// TwinCAT 3 PLC project M1_CompPP
// ProgramVersion: 3.1.4023.0
// libraries:
//   Tc2_Standard, * (Beckhoff Automation GmbH)
//   Tc2_System, * (Beckhoff Automation GmbH)
//   Tc2_Utilities, * (Beckhoff Automation GmbH)
//   Tc3_EventLogger, * (Beckhoff Automation GmbH)
//   Tc3_Module, * (Beckhoff Automation GmbH)
// project tree:
//   DUTs/ E_ChargerType.TcDUT, E_State.TcDUT, E_VoltFB.TcDUT, ST_Alarm_Base.TcDUT (not stored), ST_Charger_Base.TcDUT, ST_ChargeTime.TcDUT (not stored), ST_Module.TcDUT, ST_Segment_Base.TcDUT, ST_Setpoints_Base.TcDUT, ST_VoltMon_Base.TcDUT, ST_VoltTran_Base.TcDUT (not stored)
//   GVLs/ Alarms_DB.TcGVL (not stored), ChargeTime_DB.TcGVL, EngVal.TcGVL, GVL.TcGVL (not stored), HMI_DB.TcGVL, Input.TcGVL, LCP1_IO.TcGVL, LCP2_IO.TcGVL, LCP3_IO.TcGVL, LV.TcGVL, MCP_IO.TcGVL, Output.TcGVL, Permissives_DB.TcGVL, Setpoints.TcGVL, Trips_DB.TcGVL, VoltMonitor_DB.TcGVL
//   / PlcTask.TcTTO
//   POUs/ ADC_10V.TcPOU (not stored), ADC_5V.TcPOU (not stored), Alarms.TcPOU, Alarms_FB.TcPOU, Alias.TcPOU, AnalogConversion.TcPOU, AQ.TcPOU (not stored), ChargeTime.TcPOU, Heartbeat.TcPOU (not stored), HMI.TcPOU, LCA_CAL.TcPOU (not stored), MAIN.TcPOU, Norm_x.TcPOU (not stored), Permissives.TcPOU, Stagger_FB.TcPOU, Sequence.TcPOU, VoltageMonitor.TcPOU, VoltMonAC_FB.TcPOU, VoltTranBd.TcPOU (not stored)
// real-time tasks:
//   TASK PlcTask: cycle T#10ms, priority 20, ADS port 350
// I/O:
//   DEVICE Device 1 (EtherCAT) (disabled), AmsNetId 5.107.220.56.2.1
//     Term 1 (EK1200) [EK1200-5000 EtherCAT Power supply (2A E-Bus)]
//       Term 2 (EL1008) [EL1008 8Ch. Dig. Input 24V, 3ms]
//       Term 3 (EL6695) [EL6695 EtherCAT Bridge terminal (Primary)]
//       Term 4 (EK1561) [EK1561 1 port EtherCAT junction (POF)]
//       Term 5 (EL9011) [EL9011 End Terminal]

CONFIGURATION M1_CompPP
    RESOURCE PLC ON TwinCAT3
        TASK PlcTask(INTERVAL := T#10ms, PRIORITY := 20);
        PROGRAM MAIN WITH PlcTask : MAIN;
    END_RESOURCE
END_CONFIGURATION

// ---- DUTs/E_ChargerType.TcDUT
{attribute 'qualified_only'}
{attribute 'strict'}
TYPE E_ChargerType :
(
	TDK12kV := 0,
	TDK30kV := 1,
	TDK50kV := 2
);
END_TYPE

// ---- DUTs/E_State.TcDUT
{attribute 'qualified_only'}
{attribute 'strict'}
TYPE E_State :
(
	SAFE			:= 0, //IDLE
	CHARGING		:= 1, //Charge
	CHARGECOMPLETE	:= 2, //EOC
	//DISCONNECTING	:= 3, //Disconnect
	DUMPING			:= 3, 
	ABORT			:= 4,
	TRIPPED			:= 5, 
	ManualMode		:= 6
);
END_TYPE

// ---- DUTs/E_VoltFB.TcDUT
{attribute 'qualified_only'}
{attribute 'strict'}
TYPE E_VoltFB :
(
	seg1 := 1,
	seg2 := 2,
	seg3 := 3
);
END_TYPE

// ---- DUTs/ST_Charger_Base.TcDUT
TYPE ST_Charger_Base :
STRUCT
	//DI
	inhibited 		: BOOL;
	EndOfCharge 	: BOOL;
	HV_isON			: BOOL;
	OverTemp		: BOOL;
	InterlockOpen	: BOOL;
	LoadFaulted		: BOOL;
	SummaryFaulted	: BOOL;
	
	//DQ
	inhibit			: BOOL;
	HV_ON			: BOOL;
	
	//AI
	voltageFeedback_raw 	: INT;
	voltageFeedback_norm 	: REAL;
	voltageFeedback			: REAL;
	
	currentFeedback_raw 	: INT;
	currentFeedback_norm	: REAL;
	currentFeedback			: REAL;
	
	//AQ
	voltageSP_norm	: REAL;
	voltageSP		: REAL;
	voltageSP_raw	: INT; // setpoint output to field device.
	
	//Internal
	//ChargerType_50kV : BOOL;
	//ChargerType_12kV : BOOL;
	ChargerType		 : INT;
	LossInhibit		 : BOOL;
	LossHVON		 : BOOL;
	LossInhibitTON	 : TON;
	LossHVON_TON	 : TON;
	
	ChargeTime		: ST_ChargeTime;
END_STRUCT
END_TYPE

// ---- DUTs/ST_Module.TcDUT
TYPE ST_Module :
STRUCT
	DumpRly_close	: BOOL;
	
	VoltageFeedback : ARRAY[1..2] OF REAL;
	VoltageFeedback_norm : ARRAY[1..2] OF REAL;
	VoltageFeedback_raw : ARRAY[1..2] OF DINT;
	//VTB : ARRAY[1..2] OF ST_VoltTran_Base;  uncomment this for troubleshooting the bits in VoltageMonitor POU
END_STRUCT
END_TYPE

// ---- DUTs/ST_Segment_Base.TcDUT
TYPE ST_Segment_Base :
STRUCT
	Module : ARRAY [1..9] OF ST_Module;	
	
	CloseChargeRly	: BOOL;
	ChargeRly_close : BOOL;

	OpenModule1To3DumpRly : BOOL; //Open Module1To3DumpRly
	OpenModule4To6DumpRly : BOOL;
	OpenModule7To9DumpRly : BOOL;
	
	//ShortContactClose	: BOOL;

END_STRUCT
END_TYPE

// ---- DUTs/ST_Setpoints_Base.TcDUT
TYPE ST_Setpoints_Base :
STRUCT
	RequiredChargedV : REAL := 12;
	TotalCapacitance : REAL := 10; //uF - LOCAL ONLY, NOT FROM MAIN PLC - LoadCapacitance
	PSratedV		 : REAL := 50;
	wLCA			 : BOOL := TRUE;
	NumOfCharger	 : INT := 2;
	eChargerType		: E_ChargerType;
END_STRUCT
END_TYPE

// ---- DUTs/ST_VoltMon_Base.TcDUT
TYPE ST_VoltMon_Base :
STRUCT
	VTB : ARRAY[0..24] OF ST_VoltTran_Base;
	//Heartbeat : BOOL := 0;
	(*BateryLow  : ARRAY[0..24] OF BOOL := 0;
	//Channel	: USINT; //ST_AnalogCHSelection;
	VoltageReading_raw : ARRAY[0..24] OF INT; //custom board
	VoltageReading_norm : ARRAY[0..24] OF REAL;
	//VoltageReading	: ARRAY[0..15] OF REAL;
	//LoadMaxRatedV	: REAL := 13800; //-2k TO 35kV
	//LoadMinRatedV	: REAL := -1450; //Jake's lab result
//***************************************
	CapRaw : ARRAY[0..24] OF UINT;
	CapRawBIT : ARRAY[0..24] OF STRING;
	//CapRaw_DummySnap : ARRAY[0..24] OF UINT;
	CapRaw_Str : ARRAY[0..24] OF STRING;
	
	DataNull : ARRAY[0..24] OF BOOL := 0;
	//cunter for missing packets
	missedCTU : CTU;
	//ONS	: R_TRIG;
	missingCNT : WORD :=0;
	LossVoltTransBoard : ARRAY[0..24] OF BOOL := 0;
//**********************************	
	Time1		: TON;
	Time1_ET	: TIME;
	packetsPerMin : REAL;
	//missedCTU : CTU;
	ONS	: R_TRIG;
	//missingCNT : WORD;
	missingCNT_REAL : REAL;*)
END_STRUCT
END_TYPE

// ---- GVLs/ChargeTime_DB.TcGVL
{attribute 'qualified_only'}
VAR_GLOBAL RETAIN
	ChargerDelay_TON : ARRAY[1..7] OF TON;
	ChargerDelay_PT  : ARRAY[1..7] OF TIME;
	ChargerDelay_ET  : ARRAY[1..7] OF TIME;	
	
	//SustChargeTime_TON : ARRAY[1..3] OF TON;
	//SustChargeTime_PT  : ARRAY[1..3] OF TIME;
	//SustChargeTime_ET  : ARRAY[1..3] OF TIME;	
	
	//FormChargeTime_TON : ARRAY[1..2] OF TON;
	//FormChargeTime_PT  : ARRAY[1..2] OF TIME;
	//FormChargeTime_ET  : ARRAY[1..2] OF TIME;
	
	PreFormChargeTime_TON : TON;
	PreFormChargeTime_PT : TIME;
	PreFormChargeTime_ET : TIME;
	
	LongestChargeTime_TON : TON;
	LongestChargeTime_PT : TIME;
	LongestChargeTime_ET : TIME;

	ChargeTimeStartDelay	: ARRAY[1..7] OF INT;
	ChargingTimeElapse		: ARRAY[1..7] OF INT;	
	ChargingTimeElapse_TON	: ARRAY[1..7] OF TON;
	
	PreFormChargeTimeStartDelay : INT;
	PreFormChargingTimeElapse : INT;
	PreFormChargingTimeElapse_TON : TON;
END_VAR

// ---- GVLs/EngVal.TcGVL
{attribute 'qualified_only'}
VAR_GLOBAL
	Max_50kVChargerVoltage : REAL := 50000; //50kV
	Min_50kVChargerVoltage : REAL := 0;
	
	Max_50kVChargerCurrent : REAL := 0.18; //total peak charge current is 0.18A
	Min_50kVChargerCurrent : REAL := 0;
	
	Max_12kVChargerVoltage : REAL := 12000; //12kV
	Min_12kVChargerVoltage : REAL := 0;
	
	Max_12kVChargerCurrent : REAL := 0.75; //total peak charge current is 0.75A
	Min_12kVChargerCurrent : REAL := 0;
	
	Max_30kVChargerVoltage : REAL := 30000; //30kV
	Min_30kVChargerVoltage : REAL := 0;
	
	Max_30kVChargerCurrent : REAL := 0.6; //total peak charge current is 0.6A
	Min_30kVChargerCurrent : REAL := 0;	
	//Max_GLS1_ChargerV	   : REAL := 50000; //form trigger
	//Max_GLS2_ChargerV	   : REAL := 50000; // preform trigger
	//Max_GLS3_ChargerV	   : REAL := 30000; // preform cap charger
	
	Max_CapVoltage			: REAL := 32000;  //assuming 32kV cap....  
	Min_CapVoltage			: REAL := 0;
	
	UpperLimit12kVCaps		: REAL := 10500; 
	//LowerLimit12kVCaps	: REAL := -2000;
	UpperLimit50kVCaps		: REAL := 35000; 
	
	(*ULimit_PeakCapRequiredV	: REAL := 10000; //10kV veto
	LLimit_PeakCapRequiredV	: REAL := -2000; //-2kV
	ULimit_SustCapRequiredV	: REAL := 12000; //12kv veto
	LLimit_SustCapRequiredV	: REAL := -2000; //-2kv
	ULimit_FormCapRequiredV : REAL := 35000;
	LLimit_FormCapRequiredV : REAL := 0;
	*)
	//ULimit_PreFormCapRequiredV : REAL := 30000; //gls3
	//LLimit_PreFormCapRequiredV : REAL := 0;
		
END_VAR

// ---- GVLs/HMI_DB.TcGVL
{attribute 'qualified_only'}
VAR_GLOBAL PERSISTENT
	TDKLoad		: ARRAY [1..7] OF ST_Setpoints_Base; //or RETAIN
	
	ChargerHVOFF_rlyDelayPT		: TIME := T#25MS;
	ChargerHVOFF_rlyDelayPT_INT	: INT := 25;
	
	HVONdelayPT					: TIME := T#250MS;
	HVONdelayPT_INT				: INT := 250;
	
	RunOutTMR_PT				: TIME := T#10S;
	RunOutTMR_PT_INT			: DINT := 10;
	RunOutTMR_elapse			: DINT;
	
	ChargingRunOutTMR_elapse	: INT;

END_VAR

VAR_GLOBAL
	ChargePB					: BOOL := 0;
	DumpPB						: BOOL := 0;
	AbortPB						: BOOL := 0;
	FirePB						: BOOL := 0;
	ClearFaultPB				: BOOL := 0;
	AllDumpRelaysOpenBP			: BOOL := 0;
	AllDumpRelaysCloseBP		: BOOL := 0;
	AllCapsDischargedBP			: BOOL := 0;
	AllChargeRelayCloseBP		: BOOL := 0;
	AllVoltMonBoardStatusOKBP	: BOOL := 0;
	SystemSafeBP				: BOOL := 0;
	
	HMI_ManualModeSelected		: BOOL := 0;  // 1 = manual mode selected
	CloseChargeRlySW			: BOOL := 0;
	OpenDumpRlySW				: BOOL := 0;
	TurnChrgHVonSW				: BOOL := 0;
	TurnChrgInhibitOffSW		: BOOL := 0;
	TurnOnShotTrigSW			: BOOL := 0;
	TurnOnChargeAlarm			: BOOL := 0;
	
	LastTimeShotLog				: BOOL := 0;
END_VAR

// ---- GVLs/Input.TcGVL
{attribute 'qualified_only'}
VAR_GLOBAL
//***MCP************************************************************************
	//EL1008 - DI1
	R1_01_00 AT	%I*: BOOL; //Master stop PB not pressed - black pb on mcp
	R1_01_01 AT	%I*: BOOL; //case Estop circuit okay (Rly1 (120vac)
	R1_01_02 AT %I*: BOOL; //MCP PSU1 DC OK
	R1_01_03 AT %I*: BOOL; //
	R1_01_04 AT %I*: BOOL; //
	R1_01_05 AT %I*: BOOL; //spare
	R1_01_06 AT %I*: BOOL; //spare
	R1_01_07 AT %I*: BOOL; //spare

	//EL1008 - DI2
	R1_02_00 AT	%I*: BOOL; 
	R1_02_01 AT	%I*: BOOL;
	R1_02_02 AT %I*: BOOL; 
	R1_02_03 AT %I*: BOOL; 
	R1_02_04 AT %I*: BOOL; 
	R1_02_05 AT %I*: BOOL; 
	R1_02_06 AT %I*: BOOL; 
	R1_02_07 AT %I*: BOOL;  
	
	//EL1008 - DI3
	R1_03_00 AT	%I*: BOOL;  
	R1_03_01 AT	%I*: BOOL;
	R1_03_02 AT %I*: BOOL; 
	R1_03_03 AT %I*: BOOL; 
	R1_03_04 AT %I*: BOOL; 
	R1_03_05 AT %I*: BOOL; 
	R1_03_06 AT %I*: BOOL; 
	R1_03_07 AT %I*: BOOL;  
	
	//EL1008 - DI4
	R1_04_00 AT	%I*: BOOL;  
	R1_04_01 AT	%I*: BOOL;
	R1_04_02 AT %I*: BOOL; 
	R1_04_03 AT %I*: BOOL; 
	R1_04_04 AT %I*: BOOL; 
	R1_04_05 AT %I*: BOOL; 
	R1_04_06 AT %I*: BOOL; 
	R1_04_07 AT %I*: BOOL; 
	
	//EL1008 - DI5
	R1_05_00 AT	%I*: BOOL;  
	R1_05_01 AT	%I*: BOOL;
	R1_05_02 AT %I*: BOOL; 
	R1_05_03 AT %I*: BOOL; 
	R1_05_04 AT %I*: BOOL; 
	R1_05_05 AT %I*: BOOL; 
	R1_05_06 AT %I*: BOOL; 
	R1_05_07 AT %I*: BOOL;
	
	//EL3068 - AI1
	R1_08_00 		AT %I*: INT;
	R1_08_00_Status AT %I*: WORD;
	
	R1_08_01 		AT %I*: INT;
	R1_08_01_Status AT %I*: WORD;

	R1_08_02 		AT %I*: INT;
	R1_08_02_Status AT %I*: WORD;

	R1_08_03 		AT %I*: INT;
	R1_08_03_Status AT %I*: WORD;

	R1_08_04 		AT %I*: INT;
	R1_08_04_Status AT %I*: WORD;

	R1_08_05 		AT %I*: INT;
	R1_08_05_Status AT %I*: WORD;

	R1_08_06 		AT %I*: INT;
	R1_08_06_Status AT %I*: WORD;

	R1_08_07 		AT %I*: INT;
	R1_08_07_Status AT %I*: WORD;

//RACK 2
	//EL3068 - AI1
	R2_01_00 		AT %I*: INT;
	R2_01_00_Status AT %I*: WORD;

	R2_01_01 		AT %I*: INT;
	R2_01_01_Status AT %I*: WORD;

	R2_01_02 		AT %I*: INT;
	R2_01_02_Status AT %I*: WORD;

	R2_01_03 		AT %I*: INT;
	R2_01_03_Status AT %I*: WORD;

	R2_01_04 		AT %I*: INT;
	R2_01_04_Status AT %I*: WORD;

	R2_01_05 		AT %I*: INT;
	R2_01_05_Status AT %I*: WORD;

	R2_01_06 		AT %I*: INT;
	R2_01_06_Status AT %I*: WORD;

	R2_01_07 		AT %I*: INT;
	R2_01_07_Status AT %I*: WORD;

	//EL3068 - AI2
	R2_02_00 		AT %I*: INT;
	R2_02_00_Status AT %I*: WORD;

	R2_02_01 		AT %I*: INT;
	R2_02_01_Status AT %I*: WORD;

	R2_02_02 		AT %I*: INT;
	R2_02_02_Status AT %I*: WORD;

	R2_02_03 		AT %I*: INT;
	R2_02_03_Status AT %I*: WORD;

	R2_02_04 		AT %I*: INT;
	R2_02_04_Status AT %I*: WORD;

	R2_02_05 		AT %I*: INT;
	R2_02_05_Status AT %I*: WORD;

	R2_02_06 		AT %I*: INT;
	R2_02_06_Status AT %I*: WORD;

	R2_02_07 		AT %I*: INT;
	R2_02_07_Status AT %I*: WORD;

	//EL1008 - DI1
	R2_03_00 AT	%I*: BOOL;  
	R2_03_01 AT	%I*: BOOL;
	R2_03_02 AT %I*: BOOL; 
	R2_03_03 AT %I*: BOOL; 
	R2_03_04 AT %I*: BOOL; 
	R2_03_05 AT %I*: BOOL; 
	R2_03_06 AT %I*: BOOL; 
	R2_03_07 AT %I*: BOOL;  

	//EL1008 - DI2
	R2_04_00 AT	%I*: BOOL;  
	R2_04_01 AT	%I*: BOOL;
	R2_04_02 AT %I*: BOOL; 
	R2_04_03 AT %I*: BOOL; 
	R2_04_04 AT %I*: BOOL; 
	R2_04_05 AT %I*: BOOL; 
	R2_04_06 AT %I*: BOOL; 
	R2_04_07 AT %I*: BOOL;  

	//EL1008 - DI3
	R2_05_00 AT	%I*: BOOL;  
	R2_05_01 AT	%I*: BOOL;
	R2_05_02 AT %I*: BOOL; 
	R2_05_03 AT %I*: BOOL; 
	R2_05_04 AT %I*: BOOL; 
	R2_05_05 AT %I*: BOOL; 
	R2_05_06 AT %I*: BOOL; 
	R2_05_07 AT %I*: BOOL;  

//Rack 3	
	//EL3068 - AI1
	R3_01_00 		AT %I*: INT;
	R3_01_00_Status AT %I*: WORD;

	R3_01_01 		AT %I*: INT;
	R3_01_01_Status AT %I*: WORD;

	R3_01_02 		AT %I*: INT;
	R3_01_02_Status AT %I*: WORD;

	R3_01_03 		AT %I*: INT;
	R3_01_03_Status AT %I*: WORD;

	R3_01_04 		AT %I*: INT;
	R3_01_04_Status AT %I*: WORD;

	R3_01_05 		AT %I*: INT;
	R3_01_05_Status AT %I*: WORD;

	R3_01_06 		AT %I*: INT;
	R3_01_06_Status AT %I*: WORD;

	R3_01_07 		AT %I*: INT;
	R3_01_07_Status AT %I*: WORD;

	//EL3068 - AI2
	R3_02_00 		AT %I*: INT;
	R3_02_00_Status AT %I*: WORD;

	R3_02_01 		AT %I*: INT;
	R3_02_01_Status AT %I*: WORD;

	R3_02_02 		AT %I*: INT;
	R3_02_02_Status AT %I*: WORD;

	R3_02_03 		AT %I*: INT;
	R3_02_03_Status AT %I*: WORD;

	R3_02_04 		AT %I*: INT;
	R3_02_04_Status AT %I*: WORD;

	R3_02_05 		AT %I*: INT;
	R3_02_05_Status AT %I*: WORD;

	R3_02_06 		AT %I*: INT;
	R3_02_06_Status AT %I*: WORD;

	R3_02_07 		AT %I*: INT;
	R3_02_07_Status AT %I*: WORD;

	//EL1008 - DI1
	R3_03_00 AT	%I*: BOOL;  
	R3_03_01 AT	%I*: BOOL;
	R3_03_02 AT %I*: BOOL; 
	R3_03_03 AT %I*: BOOL; 
	R3_03_04 AT %I*: BOOL; 
	R3_03_05 AT %I*: BOOL; 
	R3_03_06 AT %I*: BOOL; 
	R3_03_07 AT %I*: BOOL;  

	//EL1008 - DI2
	R3_04_00 AT	%I*: BOOL;  
	R3_04_01 AT	%I*: BOOL;
	R3_04_02 AT %I*: BOOL; 
	R3_04_03 AT %I*: BOOL; 
	R3_04_04 AT %I*: BOOL; 
	R3_04_05 AT %I*: BOOL; 
	R3_04_06 AT %I*: BOOL; 
	R3_04_07 AT %I*: BOOL;  

	//EL1008 - DI3
	R3_05_00 AT	%I*: BOOL;  
	R3_05_01 AT	%I*: BOOL;
	R3_05_02 AT %I*: BOOL; 
	R3_05_03 AT %I*: BOOL; 
	R3_05_04 AT %I*: BOOL; 
	R3_05_05 AT %I*: BOOL; 
	R3_05_06 AT %I*: BOOL; 
	R3_05_07 AT %I*: BOOL; 
	
	//Ethercat Device Voltage - subject to change because the VM board is still under development
	B170357_CapRaw AT %I* : ARRAY[0..24] OF UINT;
	B170357_BatLevel AT %I* : BOOL;
	B170357_Heartbeat AT %I* : BOOL;
	
	B170357_2_CapRaw AT %I* : ARRAY[0..24] OF UINT;
	B170357_2_BatLevel AT %I* : BOOL;
	B170357_2_Heartbeat AT %I* : BOOL;
	
	//Ract 4 - Shaft ramp
	//EL1008 - DI 1
	R4_01_00 AT %I*: BOOL; 
	R4_01_01 AT	%I*: BOOL;
	R4_01_02 AT %I*: BOOL; 
	R4_01_03 AT %I*: BOOL; 
	R4_01_04 AT %I*: BOOL; 
	R4_01_05 AT %I*: BOOL; 
	R4_01_06 AT %I*: BOOL; 
	R4_01_07 AT %I*: BOOL; 
	
	B170357_3_CapRaw AT %I* : ARRAY[0..24] OF UINT;  // might be 8 fruit stands so 0..7
	B170357_3_BatLevel AT %I* : BOOL;
	B170357_3_Heartbeat AT %I* : BOOL;
	
END_VAR

// ---- GVLs/LCP1_IO.TcGVL
{attribute 'qualified_only'}
VAR_GLOBAL
	Segment	: ARRAY [1..3] OF ST_Segment_Base;
	
	Segment1to3_ShortContactClose	: BOOL;
	Segment1to3_UnShortContactClose	: BOOL;
	LossInterlockPressure			: BOOL;
	PSU1OK							: BOOL;
	
	VMB : ST_VoltMon_Base;
	//VTB : ARRAY[0..17] OF ST_VoltTran_Base; 
	Fire			: BOOL;
	SegmentCharged	: BOOL;
	TriggerScope	: BOOL;
END_VAR

// ---- GVLs/LCP2_IO.TcGVL
{attribute 'qualified_only'}
VAR_GLOBAL
	Segment	: ARRAY [4..6] OF ST_Segment_Base;
	
	Segment4to6_ShortContactClose	: BOOL;
	Segment4to6_UnShortContactClose	: BOOL;
	LossInterlockPressure			: BOOL;
	PSU1OK							: BOOL;
	
	VMB : ST_VoltMon_Base;
	Fire			: BOOL;
	SegmentCharged	: BOOL;
	TriggerScope	: BOOL;
END_VAR

// ---- GVLs/LCP3_IO.TcGVL
{attribute 'qualified_only'}
VAR_GLOBAL
	//Shaft Ramp Supply
	PSU1_OK				: BOOL := FALSE;
	VMB 				: ST_VoltMon_Base;
	SegmentCharged		: BOOL := FALSE;
	CloseSRChargeRly	: BOOL := FALSE;
	SRChargeRly_close 	: BOOL := FALSE;
	OpenSRDumpRly		: ARRAY[1..8] OF BOOL;
	SRDumpRelay_close 	: BOOL := FALSE;
END_VAR

// ---- GVLs/LV.TcGVL
{attribute 'qualified_only'}
VAR_GLOBAL
	TxWord1	: WORD;
	TxWord2 : WORD;
	TxWord3 : WORD;
	
	RxWord1 : WORD;
	RxWord2 : WORD;
	RxWord3 : WORD;

	
	TxInt : ARRAY [1..5] OF INT;
	TxDint : ARRAY [1..3] OF DINT;
	TxREAL : ARRAY [1..6] OF REAL;

	RxInt : ARRAY [1..2] OF INT;
	RxDint : ARRAY [1..3] OF DINT;
	RxREAL : ARRAY [1..44] OF REAL;
	
	Charger : ARRAY[1..6] OF ST_Charger_Base;
	
	TDKLoad	: ARRAY [1..6] OF ST_Setpoints_Base; 
	
	(*ChargerHVOFF_rlyDelayPT		: TIME := T#25MS;
	ChargerHVOFF_rlyDelayPT_INT	: INT := 25;
	
	HVONdelayPT					: TIME := T#250MS;
	HVONdelayPT_INT				: INT := 250;
	
	RunOutTMR_PT				: TIME := T#10S;
	RunOutTMR_PT_INT			: DINT := 10;
	RunOutTMR_elapse			: DINT;
	
	ChargingRunOutTMR_elapse	: INT;
	
	ChargePB					: BOOL := 0;
	DumpPB						: BOOL := 0;
	AbortPB						: BOOL := 0;
	FirePB						: BOOL := 0;
	ClearFaultPB				: BOOL := 0;
	AllDumpRelaysOpenBP			: BOOL := 0;
	AllChargeRelayCloseBP		: BOOL := 0;
	SystemSafeBP				: BOOL := 0;
	
	HMI_ManualModeSelected		: BOOL := 0;  // 1 = manual mode selected
	CloseChargeRlySW			: BOOL := 0;
	OpenDumpRlySW				: BOOL := 0;*)
END_VAR

// ---- GVLs/MCP_IO.TcGVL
{attribute 'qualified_only'}
VAR_GLOBAL
	MasterStopPB_NotPressed		: BOOL;
	CageEstopCircuitOK			: BOOL;
	//RemoteModeSelected			: BOOL;
	PSU1_DCOK					: BOOL;
	//MachineGNDrlyOpen			: BOOL;
	//CloseAllChargeRlyCommand	: BOOL; only for slim
	//OpenAllDumpRelayCommand		: BOOL; only for slim
	//Charger 					: ARRAY [1..8] OF ST_Charger_Base;
	//GLS3_Load					: ST_ChargeTime;
	//GLS1_hvON					: BOOL;
	//GLS2_hvON					: BOOL;
	//GLS3_hvON					: BOOL;
	//LiftMachineGND				: BOOL;
	//AllChargeRelaysClose		: BOOL; only for slim
	//AllDumpRelaysOpen			: BOOL; only for slim
	//GLS1_voltageSP				: DINT;
	//GLS1_voltageSP_norm			: REAL;
	//GLS1_voltageSP_raw			: INT;
	
	//GLS2_voltageSP				: DINT;
	//GLS2_voltageSP_norm			: REAL;
	//GLS2_voltageSP_raw			: INT;
	
	//GLS3_voltageSP				: DINT;
	//GLS3_voltageSP_norm			: REAL;
	//GLS3_voltageSP_raw			: INT;

END_VAR

VAR_GLOBAL PERSISTENT
	Charger 					: ARRAY [1..7] OF ST_Charger_Base;
END_VAR

// ---- GVLs/Output.TcGVL
{attribute 'qualified_only'}
VAR_GLOBAL
//***MCP 
	//EL2008 - DQ1
	R1_06_00 AT %Q*: BOOL;
	R1_06_01 AT %Q*: BOOL;
	R1_06_02 AT %Q*: BOOL;
	R1_06_03 AT %Q*: BOOL;
	R1_06_04 AT %Q*: BOOL;
	R1_06_05 AT %Q*: BOOL;
	R1_06_06 AT %Q*: BOOL;
	R1_06_07 AT %Q*: BOOL;

	//EL2008 - DQ2
	R1_07_00 AT %Q*: BOOL;
	R1_07_01 AT %Q*: BOOL;
	R1_07_02 AT %Q*: BOOL;
	R1_07_03 AT %Q*: BOOL;
	R1_07_04 AT %Q*: BOOL;
	R1_07_05 AT %Q*: BOOL;
	R1_07_06 AT %Q*: BOOL;
	R1_07_07 AT %Q*: BOOL;
	
	//EL4008 - AQ1
	R1_09_00 AT %Q*: INT;	//Charger 1 - Voltage Setpoint
	R1_09_01 AT %Q*: INT;	//Charger 2 - Voltage Setpoint
	R1_09_02 AT %Q*: INT;	//Charger 3 - Voltage Setpoint
	R1_09_03 AT %Q*: INT;	//Charger 4 - Voltage Setpoint
	R1_09_04 AT %Q*: INT;	//Charger 5 - Voltage Setpoint	
	R1_09_05 AT %Q*: INT;	//Charger 6 - Voltage Setpoint	
	R1_09_06 AT %Q*: INT;	//spare
	R1_09_07 AT %Q*: INT;	//spare
	
//**LCP1
	//EL2008 - DQ1
	R2_06_00 AT %Q*: BOOL;
	R2_06_01 AT %Q*: BOOL;
	R2_06_02 AT %Q*: BOOL;
	R2_06_03 AT %Q*: BOOL;
	R2_06_04 AT %Q*: BOOL;
	R2_06_05 AT %Q*: BOOL;
	R2_06_06 AT %Q*: BOOL;
	R2_06_07 AT %Q*: BOOL;
	
	//EL2008 - DQ2
	R2_07_00 AT %Q*: BOOL;
	R2_07_01 AT %Q*: BOOL;
	R2_07_02 AT %Q*: BOOL;
	R2_07_03 AT %Q*: BOOL;
	R2_07_04 AT %Q*: BOOL;
	R2_07_05 AT %Q*: BOOL;
	R2_07_06 AT %Q*: BOOL;
	R2_07_07 AT %Q*: BOOL;

//**LCP2
	//EL2008 - DQ1
	R3_06_00 AT %Q*: BOOL;
	R3_06_01 AT %Q*: BOOL;
	R3_06_02 AT %Q*: BOOL;
	R3_06_03 AT %Q*: BOOL;
	R3_06_04 AT %Q*: BOOL;
	R3_06_05 AT %Q*: BOOL;
	R3_06_06 AT %Q*: BOOL;
	R3_06_07 AT %Q*: BOOL;
	
	//EL2008 - DQ2
	R3_07_00 AT %Q*: BOOL;
	R3_07_01 AT %Q*: BOOL;
	R3_07_02 AT %Q*: BOOL;
	R3_07_03 AT %Q*: BOOL;
	R3_07_04 AT %Q*: BOOL;
	R3_07_05 AT %Q*: BOOL;
	R3_07_06 AT %Q*: BOOL;
	R3_07_07 AT %Q*: BOOL;
	
//**LCP3
	//EL2008 - DQ 1
	R4_02_00 AT %Q*: BOOL; 
	R4_02_01 AT	%Q*: BOOL; 
	R4_02_02 AT %Q*: BOOL; 
	R4_02_03 AT %Q*: BOOL; 
	R4_02_04 AT %Q*: BOOL; 
	R4_02_05 AT %Q*: BOOL; 
	R4_02_06 AT %Q*: BOOL; 
	R4_02_07 AT %Q*: BOOL; 
	//EL2008 - DQ2
	R4_03_00 AT %Q*: BOOL; 
	R4_03_01 AT	%Q*: BOOL; 
	R4_03_02 AT %Q*: BOOL; 
	R4_03_03 AT %Q*: BOOL; 
	R4_03_04 AT %Q*: BOOL; 
	R4_03_05 AT %Q*: BOOL; 
	R4_03_06 AT %Q*: BOOL; 
	R4_03_07 AT %Q*: BOOL; 	
END_VAR

// ---- GVLs/Permissives_DB.TcGVL
{attribute 'qualified_only'}
VAR_GLOBAL
	//SafetyOK				: BOOL;
	AllChargeRelayClosed 	: BOOL := 0;
	AllDumpRelayOpen		: BOOL := 0;
	//AllDumpRelayClose		: BOOL := 0;
	ReadyToCharge			: BOOL := 0;
	AllChargerEOC			: BOOL := 0;
	
	ChargerVBelowThres		: BOOL := 0;
	ChargerVThres			: REAL := 40;
	AllChargerHVisOFF		: BOOL := 0;
	AllChargerInhibitON		: BOOL := 0;

	AllCapsDischarged		: BOOL := 0;
	CapVoltageThres			: REAL := 40;
	
	AnyLCP1MonBoardLoss		: BOOL := 0;
	AnyLCP1MonBoardBatLo	: BOOL := 0;
	AnyLCP2MonBoardLoss		: BOOL := 0;
	AnyLCP2MonBoardBatLo	: BOOL := 0;
	
	AnyVoltMonBoardLoss		: BOOL := 0;
	AnyVoltMonBoardBatLo	: BOOL := 0;
	AllVoltMonBoardStatusOK : BOOL := 0;
	SystemIsSafe			: BOOL := 0;
END_VAR

// ---- GVLs/Setpoints.TcGVL
{attribute 'qualified_only'}
VAR_GLOBAL
	TDKLoad : ARRAY [1..7] OF ST_Setpoints_Base;
	
END_VAR

// ---- GVLs/Trips_DB.TcGVL
{attribute 'qualified_only'}
VAR_GLOBAL
		
	AnyEstopPressed 			: BOOL; //might not need
	MasterSTOPPressed			: BOOL;
	AllDCpsuOK					: BOOL;
	CageDoorNotClose			: BOOL; // might not need
	//AnyChargerOverTemp			: BOOL;
	//AnyChargerLoadFault			: BOOL;
	//AnyChargerInterlockOpen		: BOOL;
	//AnyChargerFaulted			: BOOL; // same as summary fault
	
	//SystemTripped 				: BOOL;
	//InstrumentationFaulted		: BOOL;
	//AnyChargeRlyFail			: BOOL;
	//AnyDumpRlyFail				: BOOL;
	//AnyACInterlockFail			: BOOL;
	//AnyLossInhibitSignal		: BOOL;
	//AnyLossHVONsignal			: BOOL;
	
	ChargingTimerRunout         : BOOL;
	ChargedTimerRunout			: BOOL;
	DumpTimerRunout				: BOOL;
	//SystemTimeOut				: BOOL;
	NoFaultDetected				: BOOL;
	TimerRunOutON				: BOOL;
	ChargerSummaryFault			: BOOL;
	ShortingSystemUnknown		: BOOL;
END_VAR

// ---- GVLs/VoltMonitor_DB.TcGVL
{attribute 'qualified_only'}
VAR_GLOBAL
	//VoltMonDB : ARRAY [1..2] OF ST_VoltMon_Base; 
END_VAR

// ---- POUs/MAIN.TcPOU
PROGRAM MAIN
VAR
END_VAR

Alias();
Permissives();
ChargeTime();
AnalogConversion();
VoltageMonitor();
Sequence();
HMI();
Alarms();
Heartbeat();

END_PROGRAM

// ---- POUs/Alias.TcPOU
PROGRAM Alias
VAR
	i : INT := 1;
	n : INT := 7;
	a : INT := 0; //0-15
	k : INT := 0;
	m : INT := 0;
	p : INT := 0;
END_VAR

//R1 : MCP**  
	//INPUT
	//DI
	MCP_IO.MasterStopPB_NotPressed				:= Input.R1_01_00;  //NC - Master stop PB not pressed - black pb on mcp
	MCP_IO.CageEstopCircuitOK					:= Input.R1_01_01;  //case Estop circuit okay (Rly1 (120vac)  
	MCP_IO.PSU1_DCOK							:= Input.R1_01_02; // psu1 dc ok
	//Spare										:= Input.R1_01_03; //
	//Spare										:= Input.R1_01_04; // 
	//Spare										:= Input.R1_01_05; //  
	//Spare										:= Input.R1_01_06; //  
	//Spare										:= Input.R1_01_07; //
	
	//DI
	MCP_IO.Charger[1].inhibited					:= NOT Input.R1_02_00; //TDK802 1
	MCP_IO.Charger[1].EndOfCharge				:= NOT Input.R1_02_01; //TDK802 1
	MCP_IO.Charger[1].HV_isON					:= NOT Input.R1_02_02; //TDK802 1
	MCP_IO.Charger[1].SummaryFaulted			:= NOT Input.R1_02_03; //TDK802 1
	MCP_IO.Charger[2].inhibited					:= NOT Input.R1_02_04; //TDK802 2
	MCP_IO.Charger[2].EndOfCharge				:= NOT Input.R1_02_05; //TDK802 2
	MCP_IO.Charger[2].HV_isON					:= NOT Input.R1_02_06; //TDK802 2
	MCP_IO.Charger[2].SummaryFaulted			:= NOT Input.R1_02_07; //TDK802 2
	
	MCP_IO.Charger[3].inhibited					:= NOT Input.R1_03_00; //TDK802 3
	MCP_IO.Charger[3].EndOfCharge				:= NOT Input.R1_03_01; //TDK802 3
	MCP_IO.Charger[3].HV_isON					:= NOT Input.R1_03_02; //TDK802 3
	MCP_IO.Charger[3].SummaryFaulted			:= NOT Input.R1_03_03; //TDK802 3
	MCP_IO.Charger[4].inhibited					:= NOT Input.R1_03_04; //TDK802 4
	MCP_IO.Charger[4].EndOfCharge				:= NOT Input.R1_03_05; //TDK802 4
	MCP_IO.Charger[4].HV_isON					:= NOT Input.R1_03_06; //TDK802 4
	MCP_IO.Charger[4].SummaryFaulted			:= NOT Input.R1_03_07; //TDK802 4
	
	MCP_IO.Charger[5].inhibited					:= NOT Input.R1_04_00; //TDK802 5
	MCP_IO.Charger[5].EndOfCharge				:= NOT Input.R1_04_01; //TDK802 5
	MCP_IO.Charger[5].HV_isON					:= NOT Input.R1_04_02; //TDK802 5
	MCP_IO.Charger[5].SummaryFaulted			:= NOT Input.R1_04_03; //TDK802 5
	MCP_IO.Charger[6].inhibited					:= NOT Input.R1_04_04; //TDK802 6
	MCP_IO.Charger[6].EndOfCharge				:= NOT Input.R1_04_05; //TDK802 6
	MCP_IO.Charger[6].HV_isON					:= NOT Input.R1_04_06; //TDK802 6
	MCP_IO.Charger[6].SummaryFaulted			:= NOT Input.R1_04_07; //TDK802 6
	(*shaft ramp add below*)
	
	//DQ
	Output.R1_06_00	:= MCP_IO.Charger[1].inhibit;
	Output.R1_06_01	:= MCP_IO.Charger[1].HV_ON;
	Output.R1_06_02	:= MCP_IO.Charger[2].inhibit;
	Output.R1_06_03	:= MCP_IO.Charger[2].HV_ON;
	Output.R1_06_04	:= MCP_IO.Charger[3].inhibit;
	Output.R1_06_05	:= MCP_IO.Charger[3].HV_ON;
	Output.R1_06_06	:= MCP_IO.Charger[4].inhibit;
	Output.R1_06_07	:= MCP_IO.Charger[4].HV_ON;
	
	//DQ
	Output.R1_07_00	:= MCP_IO.Charger[5].inhibit;
	Output.R1_07_01	:= MCP_IO.Charger[5].HV_ON;
	Output.R1_07_02	:= MCP_IO.Charger[6].inhibit;
	Output.R1_07_03	:= MCP_IO.Charger[6].HV_ON;
	//Output.R1_07_04 := spare
	//Output.R1_07_05 spare
	//Output.R1_07_06 spare
	//Output.R1_07_07 spare
	
	//EL3068 - AI
	MCP_IO.Charger[1].voltageFeedback_raw		:= Input.R1_08_00;
	MCP_IO.Charger[2].voltageFeedback_raw		:= Input.R1_08_01;
	MCP_IO.Charger[3].voltageFeedback_raw		:= Input.R1_08_02;
	MCP_IO.Charger[4].voltageFeedback_raw		:= Input.R1_08_03;
	MCP_IO.Charger[5].voltageFeedback_raw		:= Input.R1_08_04;
	MCP_IO.Charger[6].voltageFeedback_raw		:= Input.R1_08_05;
	//Input.R1_08_06;
	//Input.R1_08_07;
		
	//EL4008 AQ
	Output.R1_09_00	:= MCP_IO.Charger[1].voltageSP_raw;
	Output.R1_09_01	:= MCP_IO.Charger[2].voltageSP_raw;
	Output.R1_09_02	:= MCP_IO.Charger[3].voltageSP_raw;
	Output.R1_09_03	:= MCP_IO.Charger[4].voltageSP_raw;	
	Output.R1_09_04	:= MCP_IO.Charger[5].voltageSP_raw;
	Output.R1_09_05	:= MCP_IO.Charger[6].voltageSP_raw;
	
//R2 : LCP1***********************************************	
	//EL3068 - AI
	(*
	LCP1_IO.Segment[1].Module[1].voltageFeedback_raw := Input.R2_01_00;
	LCP1_IO.Segment[1].Module[2].voltageFeedback_raw := Input.R2_01_01;
	LCP1_IO.Segment[1].Module[3].voltageFeedback_raw := Input.R2_01_02;
	LCP1_IO.Segment[2].Module[4].voltageFeedback_raw := Input.R2_01_03;
	LCP1_IO.Segment[2].Module[5].voltageFeedback_raw := Input.R2_01_04;
	LCP1_IO.Segment[2].Module[6].voltageFeedback_raw := Input.R2_01_05;
	LCP1_IO.Segment[3].Module[7].voltageFeedback_raw := Input.R2_01_06;	
	LCP1_IO.Segment[3].Module[8].voltageFeedback_raw := Input.R2_01_07;
	
	//EL3068 - AI
	LCP1_IO.Segment[3].Module[9].voltageFeedback_raw := Input.R2_02_00;
	*)
	
//voltage monitor boards - two transmitter per module.
	FOR k := 0 TO 17 BY 1 DO 
		//VoltMonitor_DB.VoltMonDB[1].CapRaw[k] := Input.B170357_CapRaw[k];
		LCP1_IO.VMB.VTB[k].CapRaw := Input.B170357_CapRaw[k]; //0-17
	END_FOR
	
	//DI 
	LCP1_IO.Segment[1].ChargeRly_close			:= Input.R2_03_00; //rly1
	LCP1_IO.Segment[2].ChargeRly_close			:= Input.R2_03_01; //rly2
	LCP1_IO.Segment[3].ChargeRly_close			:= Input.R2_03_02; //rly3
	LCP1_IO.Segment[1].Module1To3DumpRly_close	:= Input.R2_03_03; //rlym_1
	LCP1_IO.Segment[2].Module4To6DumpRly_close	:= Input.R2_03_04; //rlym_2
	LCP1_IO.Segment[3].Module7To9DumpRly_close	:= Input.R2_03_05; //rlym_3  
	//spare	:= Input.R2_03_06; //rlym_4 changed from every dump relay fb to one fb per segment
	//spare	:= Input.R2_03_07; //rlym_5
	
	//DI
	//spare	:=  Input.R2_04_00; //rlym_6
	//spare	:=  Input.R2_04_01; //rlym_7
	//spare	:=  Input.R2_04_02; //rlym_8
	//spare	:=  Input.R2_04_03; //rlym_9
	LCP1_IO.Segment1to3_ShortContactClose		:= Input.R2_04_04;
	LCP1_IO.Segment1to3_UnShortContactClose		:= Input.R2_04_05;
	LCP1_IO.LossInterlockPressure				:= Input.R2_04_06;
	LCP1_IO.PSU1OK								:= Input.R2_04_07;
	
	//DQ
	Output.R2_06_00 := LCP1_IO.Segment[1].CloseChargeRly; //RLY1
	Output.R2_06_01 := LCP1_IO.Segment[2].CloseChargeRly; //RLY2
	Output.R2_06_02 := LCP1_IO.Segment[3].CloseChargeRly; //RLY3
	Output.R2_06_03 := LCP1_IO.Segment[1].OpenModule1To3DumpRly; //RLY4
	Output.R2_06_04 := LCP1_IO.Segment[2].OpenModule4To6DumpRly; //RLY5
	Output.R2_06_05 := LCP1_IO.Segment[3].OpenModule7To9DumpRly; //RLY6
	Output.R2_06_06 := LCP1_IO.Fire; //opto1
	Output.R2_06_07 := LCP1_IO.SegmentCharged; //LED

//R3 : LCP2***********************************************	
	//EL3068 - AI
	(*
	LCP2_IO.Segment[4].Module[1].voltageFeedback_raw := Input.R3_01_00;
	LCP2_IO.Segment[4].Module[2].voltageFeedback_raw := Input.R3_01_01;
	LCP2_IO.Segment[4].Module[3].voltageFeedback_raw := Input.R3_01_02;
	LCP2_IO.Segment[5].Module[4].voltageFeedback_raw := Input.R3_01_03;
	LCP2_IO.Segment[5].Module[5].voltageFeedback_raw := Input.R3_01_04;
	LCP2_IO.Segment[5].Module[6].voltageFeedback_raw := Input.R3_01_05;
	LCP2_IO.Segment[6].Module[7].voltageFeedback_raw := Input.R3_01_06;	
	LCP2_IO.Segment[6].Module[8].voltageFeedback_raw := Input.R3_01_07;
	
	//EL3068 - AI
	LCP2_IO.Segment[6].Module[9].voltageFeedback_raw := Input.R3_02_00;
	*)
//voltage monitor boards - two transmitter per module.
	FOR k := 0 TO 17 BY 1 DO 
		 LCP2_IO.VMB.VTB[k].CapRaw := Input.B170357_2_CapRaw[k];
	END_FOR
	
	//DI 
	LCP2_IO.Segment[4].ChargeRly_close			:= Input.R3_03_00; //rly1
	LCP2_IO.Segment[5].ChargeRly_close			:= Input.R3_03_01; //rly2
	LCP2_IO.Segment[6].ChargeRly_close			:= Input.R3_03_02; //rly3
	LCP2_IO.Segment[4].Module1To3DumpRly_close	:= Input.R3_03_03;
	LCP2_IO.Segment[5].Module4To6DumpRly_close	:= Input.R3_03_04;
	LCP2_IO.Segment[6].Module7To9DumpRly_close	:= Input.R3_03_05;
	//spare	:= Input.R3_03_06;
	//spare	:= Input.R3_03_07;
	
	//DI
	//spare	:= Input.R3_04_00;
	//spare	:= Input.R3_04_01;
	//spare	:= Input.R3_04_02;
	//spare	:= Input.R3_04_03;
	LCP2_IO.Segment4to6_ShortContactClose		:= Input.R3_04_04;
	LCP2_IO.Segment4to6_UnShortContactClose		:= Input.R3_04_05;
	LCP2_IO.LossInterlockPressure				:= Input.R3_04_06;
	LCP2_IO.PSU1OK								:= Input.R3_04_07;
	
	//DQ
	Output.R3_06_00 := LCP2_IO.Segment[4].CloseChargeRly; //RLY1
	Output.R3_06_01 := LCP2_IO.Segment[5].CloseChargeRly; //RLY2
	Output.R3_06_02 := LCP2_IO.Segment[6].CloseChargeRly; //RLY3
	Output.R3_06_03 := LCP2_IO.Segment[4].OpenModule1To3DumpRly; //RLY4
	Output.R3_06_04 := LCP2_IO.Segment[5].OpenModule4To6DumpRly; //RLY5
	Output.R3_06_05 := LCP2_IO.Segment[6].OpenModule7To9DumpRly; //RLY6
	Output.R3_06_06 := LCP2_IO.Fire; //opto1
	Output.R3_06_07 := LCP2_IO.SegmentCharged; //LED

//R4 : LCP 3 
	//DI
	LCP3_IO.PSU1_OK					:= Input.R4_01_00;
	LCP3_IO.SRChargeRly_close		:= Input.R4_01_01;
	LCP3_IO.SRDumpRelay_close		:= Input.R4_01_02;
	
	//DQ
	Output.R4_02_00				:= LCP3_IO.CloseSRChargeRly;
	Output.R4_02_01				:= LCP3_IO.OpenSRDumpRly[1];
	Output.R4_02_02				:= LCP3_IO.OpenSRDumpRly[2];
	Output.R4_02_03				:= LCP3_IO.OpenSRDumpRly[3];
	Output.R4_02_04				:= LCP3_IO.OpenSRDumpRly[4];
	Output.R4_02_05				:= LCP3_IO.OpenSRDumpRly[5];
	Output.R4_02_06				:= LCP3_IO.OpenSRDumpRly[6];
	Output.R4_02_07				:= LCP3_IO.OpenSRDumpRly[7];
	
	Output.R4_03_00				:= LCP3_IO.OpenSRDumpRly[8];
	
	// need to have how many voltage monitor board or voltage transmitter board per fruit stand ????
	//LCP3_IO.VMB.VTB[1].

	//LV Alias
	//commented out to test the sequence
	(*
	HMI_DB.ChargePB 				:= LV.TxWord1.0;
	HMI_DB.DumpPB					:= LV.TxWord1.1;		
	HMI_DB.AbortPB					:= LV.TxWord1.2;
	HMI_DB.FirePB					:= LV.TxWord1.3;
	HMI_DB.ClearFaultPB 			:= LV.TxWord1.4;
	HMI_DB.AllDumpRelaysOpenBP		:= LV.TxWord1.5;
	HMI_DB.AllChargeRelayCloseBP	:= LV.TxWord1.6;
	HMI_DB.SystemSafeBP				:= LV.TxWord1.7;
	HMI_DB.CloseChargeRlySW			:= LV.TxWord1.8;
	HMI_DB.OpenDumpRlySW 			:= LV.TxWord1.9;
	HMI_DB.HMI_ManualModeSelected	:= LV.TxWord1.10;  // 1 = manual mode selected
	HMI_DB.TurnChrgHVonSW			:= LV.TxWord1.11;
	HMI_DB.TurnChrgInhibitOffSW		:= LV.TxWord1.12;
	HMI_DB.TurnOnShotTrigSW			:= LV.TxWord1.13;
	HMI_DB.TurnOnChargeAlarm		:= LV.TxWord1.14;
	HMI_DB.AllVoltMonBoardStatusOKBP:= LV.TxWord1.15;
	//not sure if you want to control these via LV
	(*
	MCP_IO.Charger[1].HV_ON			:= LV.TxWord2.0;
	MCP_IO.Charger[1].inhibit		:= LV.TxWord2.1;
	MCP_IO.Charger[2].HV_ON			:= LV.TxWord2.2;
	MCP_IO.Charger[2].inhibit		:= LV.TxWord2.3;
	
	MCP_IO.Charger[3].HV_ON			:= LV.TxWord2.4;
	MCP_IO.Charger[3].inhibit		:= LV.TxWord2.5;
	MCP_IO.Charger[4].HV_ON			:= LV.TxWord2.6;
	MCP_IO.Charger[4].inhibit		:= LV.TxWord2.7;
	MCP_IO.Charger[5].HV_ON			:= LV.TxWord2.8;
	MCP_IO.Charger[5].inhibit		:= LV.TxWord2.9;
	MCP_IO.Charger[6].HV_ON			:= LV.TxWord2.10;
	MCP_IO.Charger[6].inhibit		:= LV.TxWord2.11;
	HMI_DB.HMI_DB.AllDumpRelaysCloseBP := LV.TxWord2.12;
	*)
	
	LV.RxWord1.0 := LV.Charger[1].EndOfCharge			:= MCP_IO.Charger[1].EndOfCharge;
	LV.RxWord1.1 := LV.Charger[1].HV_isON				:= MCP_IO.Charger[1].HV_isON;
	LV.RxWord1.2 := LV.Charger[1].inhibited				:= MCP_IO.Charger[1].inhibited;
	LV.RxWord1.3 := LV.Charger[1].SummaryFaulted		:= MCP_IO.Charger[1].SummaryFaulted;
	LV.RxWord1.4 := LV.Charger[2].EndOfCharge			:= MCP_IO.Charger[2].EndOfCharge;
	LV.RxWord1.5 := LV.Charger[2].HV_isON				:= MCP_IO.Charger[2].HV_isON;
	LV.RxWord1.6 := LV.Charger[2].inhibited				:= MCP_IO.Charger[2].inhibited;
	LV.RxWord1.7 := LV.Charger[2].SummaryFaulted		:= MCP_IO.Charger[2].SummaryFaulted;
	LV.RxWord1.8 := LV.Charger[3].EndOfCharge			:= MCP_IO.Charger[3].EndOfCharge;
	LV.RxWord1.9 := LV.Charger[3].HV_isON				:= MCP_IO.Charger[3].HV_isON;
	LV.RxWord1.10 := LV.Charger[3].inhibited			:= MCP_IO.Charger[3].inhibited;
	LV.RxWord1.11 := LV.Charger[3].SummaryFaulted		:= MCP_IO.Charger[3].SummaryFaulted;
	LV.RxWord1.12 := LV.Charger[4].EndOfCharge			:= MCP_IO.Charger[4].EndOfCharge;
	LV.RxWord1.13 := LV.Charger[4].HV_isON				:= MCP_IO.Charger[4].HV_isON;
	LV.RxWord1.14 := LV.Charger[4].inhibited			:= MCP_IO.Charger[4].inhibited;
	LV.RxWord1.15 := LV.Charger[4].SummaryFaulted		:= MCP_IO.Charger[4].SummaryFaulted;
	
	LV.RxWord2.0 := LV.Charger[5].EndOfCharge			:= MCP_IO.Charger[5].EndOfCharge;
	LV.RxWord2.1 := LV.Charger[5].HV_isON				:= MCP_IO.Charger[5].HV_isON;
	LV.RxWord2.2 := LV.Charger[5].inhibited				:= MCP_IO.Charger[5].inhibited;
	LV.RxWord2.3 := LV.Charger[5].SummaryFaulted		:= MCP_IO.Charger[5].SummaryFaulted;
	LV.RxWord2.4 := LV.Charger[6].EndOfCharge			:= MCP_IO.Charger[6].EndOfCharge;
	LV.RxWord2.5 := LV.Charger[6].HV_isON				:= MCP_IO.Charger[6].HV_isON;
	LV.RxWord2.6 := LV.Charger[6].inhibited				:= MCP_IO.Charger[6].inhibited;
	LV.RxWord2.7 := LV.Charger[6].SummaryFaulted		:= MCP_IO.Charger[6].SummaryFaulted;
	(*shaft ramp add below*)
	
	LV.RxWord3.0 := LCP1_IO.Segment[1].ChargeRly_close;
	LV.RxWord3.1 := LCP1_IO.Segment[2].ChargeRly_close;
	LV.RxWord3.2 := LCP1_IO.Segment[3].ChargeRly_close;
	LV.RxWord3.3 := LCP2_IO.Segment[4].ChargeRly_close;
	LV.RxWord3.4 := LCP2_IO.Segment[5].ChargeRly_close;
	LV.RxWord3.5 := LCP2_IO.Segment[6].ChargeRly_close;
	
	LV.RxWord3.6 := LCP1_IO.Segment[1].Module1To3DumpRly_close;
	LV.RxWord3.7 := LCP1_IO.Segment[2].Module4To6DumpRly_close;
	LV.RxWord3.8 := LCP1_IO.Segment[3].Module7To9DumpRly_close;
	LV.RxWord3.9 := LCP2_IO.Segment[4].Module1To3DumpRly_close;
	LV.RxWord3.10 := LCP2_IO.Segment[5].Module4To6DumpRly_close;
	LV.RxWord3.11 := LCP2_IO.Segment[6].Module7To9DumpRly_close; 
	//LV.RxWord3.12  
	//LV.RxWord3.13  
	//LV.RxWord3.14  
	//LV.RxWord3.15  
	
	HMI_DB.ChargerHVOFF_rlyDelayPT_INT	:= LV.TxInt[1];
	HMI_DB.HVONdelayPT_INT 				:= LV.TxInt[2];
	LV.RxInt[1]							:= HMI_DB.ChargingRunOutTMR_elapse;
	
	HMI_DB.RunOutTMR_PT_INT				:= LV.TxDint[1];
	LV.RxDint[1]						:= HMI_DB.RunOutTMR_elapse;	
	
	
	FOR i := 1 TO n BY 1 DO
		HMI_DB.TDKLoad[i].eChargerType 					:= LV.TDKLoad[i].eChargerType;
		HMI_DB.TDKLoad[i].PSratedV						:= LV.TDKLoad[i].PSratedV;
		HMI_DB.TDKLoad[i].RequiredChargedV 				:= LV.TDKLoad[i].RequiredChargedV;
		HMI_DB.TDKLoad[i].wLCA							:= LV.TDKLoad[i].wLCA;;
		HMI_DB.TDKLoad[i].NumOfCharger					:= LV.TDKLoad[i].NumOfCharger;	
		HMI_DB.TDKLoad[i].TotalCapacitance				:= LV.TDKLoad[i].TotalCapacitance;

		LV.Charger[i].ChargeTime 						:= MCP_IO.Charger[i].ChargeTime;
		LV.RxREAL[i] := LV.Charger[i].voltageFeedback	:= MCP_IO.Charger[i].voltageFeedback; //LV.RxREAL[8] for shaft ramp
		MCP_IO.Charger[i].voltageSP (*make this real*)	:= LV.TxREAL[i] := LV.Charger[i].voltageSP;
	
	END_FOR
	
	 //lcp 1 cap volt to lv
		 LV.RxREAL[9] := LCP1_IO.Segment[1].Module[1].VoltageFeedback[1];
		 LV.RxREAL[10] := LCP1_IO.Segment[1].Module[1].VoltageFeedback[2];
		 LV.RxREAL[11] := LCP1_IO.Segment[1].Module[2].VoltageFeedback[1];
		 LV.RxREAL[12] := LCP1_IO.Segment[1].Module[2].VoltageFeedback[2];
		 LV.RxREAL[13] := LCP1_IO.Segment[1].Module[3].VoltageFeedback[1];
		 LV.RxREAL[14] := LCP1_IO.Segment[1].Module[3].VoltageFeedback[2];
		 
		 LV.RxREAL[15] := LCP1_IO.Segment[2].Module[4].VoltageFeedback[1];
		 LV.RxREAL[16] := LCP1_IO.Segment[2].Module[4].VoltageFeedback[2];
		 LV.RxREAL[17] := LCP1_IO.Segment[2].Module[5].VoltageFeedback[1];
		 LV.RxREAL[18] := LCP1_IO.Segment[2].Module[5].VoltageFeedback[2];
		 LV.RxREAL[19] := LCP1_IO.Segment[2].Module[6].VoltageFeedback[1];
		 LV.RxREAL[20] := LCP1_IO.Segment[2].Module[6].VoltageFeedback[2];
		 
		 LV.RxREAL[21] := LCP1_IO.Segment[3].Module[7].VoltageFeedback[1];
		 LV.RxREAL[22] := LCP1_IO.Segment[3].Module[7].VoltageFeedback[2];
		 LV.RxREAL[23] := LCP1_IO.Segment[3].Module[8].VoltageFeedback[1];
		 LV.RxREAL[24] := LCP1_IO.Segment[3].Module[8].VoltageFeedback[2];
		 LV.RxREAL[25] := LCP1_IO.Segment[3].Module[9].VoltageFeedback[1];
		 LV.RxREAL[26] := LCP1_IO.Segment[3].Module[9].VoltageFeedback[2];
		 
	//lcp2 cap volt to lv	 
		 LV.RxREAL[27] := LCP2_IO.Segment[4].Module[1].VoltageFeedback[1];
		 LV.RxREAL[28] := LCP2_IO.Segment[4].Module[1].VoltageFeedback[2];
		 LV.RxREAL[29] := LCP2_IO.Segment[4].Module[2].VoltageFeedback[1];
		 LV.RxREAL[30] := LCP2_IO.Segment[4].Module[2].VoltageFeedback[2];
		 LV.RxREAL[31] := LCP2_IO.Segment[4].Module[3].VoltageFeedback[1];
		 LV.RxREAL[32] := LCP2_IO.Segment[4].Module[3].VoltageFeedback[2];
		
		 LV.RxREAL[33] := LCP2_IO.Segment[5].Module[4].VoltageFeedback[1];
		 LV.RxREAL[34] := LCP2_IO.Segment[5].Module[4].VoltageFeedback[2];
		 LV.RxREAL[35] := LCP2_IO.Segment[5].Module[5].VoltageFeedback[1];
		 LV.RxREAL[36] := LCP2_IO.Segment[5].Module[5].VoltageFeedback[2];
		 LV.RxREAL[37] := LCP2_IO.Segment[5].Module[6].VoltageFeedback[1];
		 LV.RxREAL[38] := LCP2_IO.Segment[5].Module[6].VoltageFeedback[2];
		 
		 LV.RxREAL[39] := LCP2_IO.Segment[6].Module[7].VoltageFeedback[1];
		 LV.RxREAL[40] := LCP2_IO.Segment[6].Module[7].VoltageFeedback[2];
		 LV.RxREAL[41] := LCP2_IO.Segment[6].Module[8].VoltageFeedback[1];
		 LV.RxREAL[42] := LCP2_IO.Segment[6].Module[8].VoltageFeedback[2];
		 LV.RxREAL[43] := LCP2_IO.Segment[6].Module[9].VoltageFeedback[1];
		 LV.RxREAL[44] := LCP2_IO.Segment[6].Module[9].VoltageFeedback[2];
		 *)
	
IF k > 17 THEN 
	k := 0;
END_IF

IF m > 17 THEN 
	m := 0;
END_IF

IF p > 17 THEN 
	p := 0;
END_IF

IF i > n THEN 
	i := 0;
END_IF

END_PROGRAM

// ---- POUs/ChargeTime.TcPOU
PROGRAM ChargeTime
VAR

	lca_charge_cal	 : ARRAY [1..7] OF LCA_CAL;
	i				 : INT := 1; // 1-8 instances
	j				 : INT := 1; //1 - 8 ch
	m				 : INT := 1;
	n				 : INT := 7;
	a				 : INT := 1; 
	
	Q				 : REAL := 1; // Charge
	Current			 : REAL := 0.1; //100mA
	
	longestChargeTime: REAL;
	
END_VAR

//mapping hmi input to setpoints
FOR j := 1 TO n BY 1 DO	
	Setpoints.TDKLoad[j].TotalCapacitance	:= HMI_DB.TDKLoad[j].TotalCapacitance;
	Setpoints.TDKLoad[j].PSratedV 			:= HMI_DB.TDKLoad[j].PSratedV;
	Setpoints.TDKLoad[j].RequiredChargedV	:= HMI_DB.TDKLoad[j].RequiredChargedV;  
	Setpoints.TDKLoad[j].wLCA				:= HMI_DB.TDKLoad[j].wLCA;
	Setpoints.TDKLoad[j].NumOfCharger		:= HMI_DB.TDKLoad[j].NumOfCharger;	
	
	//charge time delay and elapse for HMI
	ChargeTime_DB.ChargeTimeStartDelay[j] := TIME_TO_INT((ChargeTime_DB.ChargerDelay_PT[j] - ChargeTime_DB.ChargerDelay_ET[j])/1000);
	ChargeTime_DB.ChargingTimeElapse[j] := TIME_TO_INT((ChargeTime_DB.ChargingTimeElapse_TON[j].PT - ChargeTime_DB.ChargingTimeElapse_TON[j].ET)/1000);
END_FOR

//ChargeTime_DB.PreFormChargeTimeStartDelay := TIME_TO_INT((ChargeTime_DB.PreFormChargeTime_PT - ChargeTime_DB.PreFormChargeTime_ET)/1000);
//ChargeTime_DB.PreFormChargingTimeElapse := TIME_TO_INT((ChargeTime_DB.PreFormChargingTimeElapse_TON.PT - ChargeTime_DB.PreFormChargingTimeElapse_TON.ET)/1000);

(*
//GLS 3
Setpoints.GLSLoad.TotalCapacitance	:= HMI_DB.GLSLoad.TotalCapacitance;
Setpoints.GLSLoad.PSratedV 			:= HMI_DB.GLSLoad.PSratedV;
//Setpoints.PreFormBank.RequiredChargedV	:= Recipe.PreFormBank.RequiredChargedV; //only thing that comes from the main plc recipe
//Setpoints.GLSLoad.wLCA				:= HMI_DB.GLSLoad.wLCA;
Setpoints.GLSLoad.NumOfCharger		:= HMI_DB.GLSLoad.NumOfCharger;	
*)


//veto
//this should not happen
FOR m := 1 TO n BY 1 DO
	IF Setpoints.TDKLoad[m].RequiredChargedV <= -2 THEN
		Setpoints.TDKLoad[m].RequiredChargedV := -2;
	END_IF	
END_FOR

FOR i := 1 TO n BY 1 DO
	IF MCP_IO.Charger[i].ChargerType = E_ChargerType.TDK50kV THEN 
		//set limites of charger voltage input from HMI input
		IF 1000*(Setpoints.TDKLoad[i].RequiredChargedV) >= EngVal.UpperLimit50kVCaps THEN
			Setpoints.TDKLoad[i].RequiredChargedV := (EngVal.UpperLimit50kVCaps/1000); //limit at 35kv
			HMI_DB.TDKLoad[i].RequiredChargedV := (EngVal.UpperLimit50kVCaps/1000);
		ELSIF Setpoints.TDKLoad[i].RequiredChargedV <= 0 THEN
			Setpoints.TDKLoad[i].RequiredChargedV := 0;
			HMI_DB.TDKLoad[i].RequiredChargedV := 0;
		END_IF
	ELSIF MCP_IO.Charger[i].ChargerType = E_ChargerType.TDK12kV OR MCP_IO.Charger[i].ChargerType = E_ChargerType.TDK30kV THEN
		//set limites of charger voltage input from HMI input
		IF 1000*(Setpoints.TDKLoad[i].RequiredChargedV) >= EngVal.UpperLimit12kVCaps THEN
			Setpoints.TDKLoad[i].RequiredChargedV := (EngVal.UpperLimit12kVCaps/1000); //limit at 10kv
			HMI_DB.TDKLoad[i].RequiredChargedV := (EngVal.UpperLimit12kVCaps/1000); //limit at 10kv
		ELSIF Setpoints.TDKLoad[i].RequiredChargedV <= 0 THEN
			Setpoints.TDKLoad[i].RequiredChargedV := ABS(Setpoints.TDKLoad[i].RequiredChargedV);
			HMI_DB.TDKLoad[i].RequiredChargedV := ABS(Setpoints.TDKLoad[i].RequiredChargedV);
		END_IF
	END_IF;
END_FOR;

(*//ch 1 - 3
IF Setpoints.TDKLoad[1].RequiredChargedV >= 10 THEN
	Setpoints.TDKLoad[1].RequiredChargedV := 10;
	ELSIF Setpoints.TDKLoad[1].RequiredChargedV < 0 THEN
		Setpoints.TDKLoad[1].RequiredChargedV := ABS(Setpoints.TDKLoad[1].RequiredChargedV); 
END_IF
IF Setpoints.TDKLoad[2].RequiredChargedV >= 10 THEN
	Setpoints.TDKLoad[2].RequiredChargedV := 10;
	ELSIF Setpoints.TDKLoad[2].RequiredChargedV < 0 THEN
		Setpoints.TDKLoad[2].RequiredChargedV := ABS(Setpoints.TDKLoad[2].RequiredChargedV); 	
END_IF
IF Setpoints.TDKLoad[3].RequiredChargedV >= 10 THEN
	Setpoints.TDKLoad[3].RequiredChargedV := 10;
	ELSIF Setpoints.TDKLoad[3].RequiredChargedV < 0 THEN
		Setpoints.TDKLoad[3].RequiredChargedV := ABS(Setpoints.TDKLoad[3].RequiredChargedV); 	
END_IF

//ch 4-6
IF Setpoints.TDKLoad[4].RequiredChargedV >= 12 THEN
	Setpoints.TDKLoad[4].RequiredChargedV := 12;
	ELSIF Setpoints.TDKLoad[4].RequiredChargedV < 0 THEN
		Setpoints.TDKLoad[4].RequiredChargedV := ABS(Setpoints.TDKLoad[4].RequiredChargedV); 	
END_IF
IF Setpoints.TDKLoad[5].RequiredChargedV >= 12 THEN
	Setpoints.TDKLoad[5].RequiredChargedV := 12;
	ELSIF Setpoints.TDKLoad[5].RequiredChargedV < 0 THEN
		Setpoints.TDKLoad[5].RequiredChargedV := ABS(Setpoints.TDKLoad[5].RequiredChargedV); 	
END_IF
IF Setpoints.TDKLoad[6].RequiredChargedV >= 12 THEN
	Setpoints.TDKLoad[6].RequiredChargedV := 12;
	ELSIF Setpoints.TDKLoad[6].RequiredChargedV < 0 THEN
		Setpoints.TDKLoad[6].RequiredChargedV := ABS(Setpoints.TDKLoad[6].RequiredChargedV); 	
END_IF
*)

//chg time
FOR i := 1 TO n BY 1 DO
	lca_charge_cal[i](	PSratedV := Setpoints.TDKLoad[i].PSratedV, 
						RequiredChargeV := Setpoints.TDKLoad[i].RequiredChargedV, 
						LoadCapacitance := Setpoints.TDKLoad[i].TotalCapacitance, 
						NumOfCharger := Setpoints.TDKLoad[i].NumOfCharger, 
						wLCA := Setpoints.TDKLoad[i].wLCA
						);

	MCP_IO.Charger[i].ChargeTime.timeToChargeLoad := lca_charge_cal[i].TimeToChargeLoad;
	MCP_IO.Charger[i].ChargeTime.Power := lca_charge_cal[i].RespectedPower;
	
	IF Setpoints.TDKLoad[i].RequiredChargedV = 0 THEN
		MCP_IO.Charger[i].ChargeTime.timeToChargeLoad := 0;
		MCP_IO.Charger[i].ChargeTime.Power := 0;
	END_IF
END_FOR


(*
//gls - gls3 is preform cap charger
Q := 1000* Setpoints.GLSLoad.RequiredChargedV * (Setpoints.GLSLoad.TotalCapacitance / 1000000);
MCP_IO.GLS3_Load.timeToChargeLoad := Q / Current;
MCP_IO.GLS3_Load.Power := 1000*Setpoints.GLSLoad.RequiredChargedV * Current;
*)
//find the longest charge time.  //need more work
longestChargeTime := MAX( MCP_IO.Charger[1].ChargeTime.timeToChargeLoad,
							MCP_IO.Charger[2].ChargeTime.timeToChargeLoad,
							MCP_IO.Charger[3].ChargeTime.timeToChargeLoad,
							MCP_IO.Charger[4].ChargeTime.timeToChargeLoad,
							MCP_IO.Charger[5].ChargeTime.timeToChargeLoad,
							MCP_IO.Charger[6].ChargeTime.timeToChargeLoad,
							MCP_IO.Charger[7].ChargeTime.timeToChargeLoad  //charger 7 for shaft ramp
							(*MCP_IO.Charger[8].ChargeTime.timeToChargeLoad, *)
							(*MCP_IO.GLS3_Load.timeToChargeLoad*));

ChargeTime_DB.LongestChargeTime_PT := REAL_TO_TIME (1000*longestChargeTime);

//FOR a := 1 TO 8 BY 1 DO
FOR a := 1 TO n BY 1 DO
	IF (longestChargeTime - MCP_IO.Charger[a].ChargeTime.timeToChargeLoad) >= 0 THEN
		ChargeTime_DB.ChargerDelay_PT[a] := REAL_TO_TIME (1000*(longestChargeTime - MCP_IO.Charger[a].ChargeTime.timeToChargeLoad));
		ELSE 
			ChargeTime_DB.ChargerDelay_PT[a] := REAL_TO_TIME (1000*(MCP_IO.Charger[a].ChargeTime.timeToChargeLoad - longestChargeTime));
	END_IF;		
		
	//IF (longestChargeTime - MCP_IO.Charger[a+3].ChargeTime.timeToChargeLoad) >= 0 THEN
	//	ChargeTime_DB.SustChargeTime_PT[a] := REAL_TO_TIME (1000*(longestChargeTime - MCP_IO.Charger[a+3].ChargeTime.timeToChargeLoad));	
	//END_IF;	
	
END_FOR;


(*IF (longestChargeTime - MCP_IO.Charger[7].ChargeTime.timeToChargeLoad) >= 0 THEN
	ChargeTime_DB.FormChargeTime_PT[1] := REAL_TO_TIME (1000*(longestChargeTime - MCP_IO.Charger[7].ChargeTime.timeToChargeLoad));	
END_IF;	
IF (longestChargeTime - MCP_IO.Charger[8].ChargeTime.timeToChargeLoad) >= 0 THEN
	ChargeTime_DB.FormChargeTime_PT[2] := REAL_TO_TIME (1000*(longestChargeTime - MCP_IO.Charger[8].ChargeTime.timeToChargeLoad));	
END_IF;	

IF (longestChargeTime - MCP_IO.GLS3_Load.timeToChargeLoad) >= 0 THEN
		ChargeTime_DB.PreFormChargeTime_PT := REAL_TO_TIME (1000*(longestChargeTime - MCP_IO.GLS3_Load.timeToChargeLoad));
		ELSE
			ChargeTime_DB.PreFormChargeTime_PT := REAL_TO_TIME (1000*(MCP_IO.GLS3_Load.timeToChargeLoad -longestChargeTime));
END_IF;
*)


//IF i > 8 THEN 
IF i > n THEN 
	i := 0;
END_IF

IF j > n THEN
	j := 0;
END_IF

IF m > n THEN
	m := 0;
END_IF

//IF a > 8 THEN
IF a > n THEN
	a := 1;
END_IF;

END_PROGRAM

// ---- POUs/Permissives.TcPOU
PROGRAM Permissives
VAR
	
	
END_VAR

IF (LCP1_IO.Segment[1].ChargeRly_close = TRUE AND 
	LCP1_IO.Segment[2].ChargeRly_close = TRUE AND
	LCP1_IO.Segment[3].ChargeRly_close = TRUE AND 
	LCP2_IO.Segment[4].ChargeRly_close = TRUE AND 
	LCP2_IO.Segment[5].ChargeRly_close = TRUE AND 
	LCP2_IO.Segment[6].ChargeRly_close = TRUE) OR HMI_DB.AllChargeRelayCloseBP = TRUE
	THEN 
		Permissives_DB.AllChargeRelayClosed := TRUE;
	ELSIF 
		LCP1_IO.Segment[1].ChargeRly_close = FALSE AND 
		LCP1_IO.Segment[2].ChargeRly_close = FALSE AND
		LCP1_IO.Segment[3].ChargeRly_close = FALSE AND 
		LCP2_IO.Segment[4].ChargeRly_close = FALSE AND 
		LCP2_IO.Segment[5].ChargeRly_close = FALSE AND 
		LCP2_IO.Segment[6].ChargeRly_close = FALSE
	THEN
		Permissives_DB.AllChargeRelayClosed := FALSE;
END_IF;

IF (LCP1_IO.Segment[1].Module1To3DumpRly_close = FALSE AND 
	LCP1_IO.Segment[2].Module4To6DumpRly_close = FALSE AND
	LCP1_IO.Segment[3].Module7To9DumpRly_close = FALSE AND
	
	LCP2_IO.Segment[4].Module1To3DumpRly_close = FALSE AND 
	LCP2_IO.Segment[5].Module4To6DumpRly_close = FALSE AND
	LCP2_IO.Segment[6].Module7To9DumpRly_close = FALSE) OR HMI_DB.AllDumpRelaysOpenBP = TRUE
	THEN
		Permissives_DB.AllDumpRelayOpen := TRUE;
		ELSIF
			LCP1_IO.Segment[1].Module1To3DumpRly_close = TRUE AND 
			LCP1_IO.Segment[2].Module4To6DumpRly_close = TRUE AND
			LCP1_IO.Segment[3].Module7To9DumpRly_close = TRUE AND
			LCP2_IO.Segment[4].Module1To3DumpRly_close = TRUE AND
			LCP2_IO.Segment[5].Module4To6DumpRly_close = TRUE AND
			LCP2_IO.Segment[6].Module7To9DumpRly_close = TRUE 
		THEN
			Permissives_DB.AllDumpRelayOpen := FALSE;
END_IF;

IF Permissives_DB.AllChargeRelayClosed = TRUE AND 
	Permissives_DB.AllDumpRelayOpen = TRUE AND
	(Permissives_DB.AllVoltMonBoardStatusOK= TRUE OR HMI_DB.AllVoltMonBoardStatusOKBP = TRUE)  //voltmonitor board has missing packets, so this might be sensitive and might need to bypass
	THEN
		Permissives_DB.ReadyToCharge := TRUE;
	ELSE 
		Permissives_DB.ReadyToCharge := FALSE;
END_IF

IF MCP_IO.Charger[1].voltageFeedback <= Permissives_DB.ChargerVThres AND 
	MCP_IO.Charger[2].voltageFeedback <= Permissives_DB.ChargerVThres AND 
	MCP_IO.Charger[3].voltageFeedback <= Permissives_DB.ChargerVThres AND
	MCP_IO.Charger[4].voltageFeedback <= Permissives_DB.ChargerVThres AND
	MCP_IO.Charger[5].voltageFeedback <= Permissives_DB.ChargerVThres AND
	MCP_IO.Charger[6].voltageFeedback <= Permissives_DB.ChargerVThres
	THEN
		Permissives_DB.ChargerVBelowThres := TRUE;
	ELSE
		Permissives_DB.ChargerVBelowThres := FALSE;
END_IF;

IF MCP_IO.Charger[1].HV_isON = FALSE AND 
	MCP_IO.Charger[2].HV_isON = FALSE AND 
	MCP_IO.Charger[3].HV_isON = FALSE AND
	MCP_IO.Charger[4].HV_isON = FALSE AND
	MCP_IO.Charger[5].HV_isON = FALSE AND
	MCP_IO.Charger[6].HV_isON = FALSE 
	THEN
		Permissives_DB.AllChargerHVisOFF := TRUE;
	ELSE 
		Permissives_DB.AllChargerHVisOFF := FALSE;
END_IF

IF MCP_IO.Charger[1].inhibited = TRUE AND
	MCP_IO.Charger[2].inhibited = TRUE AND
	MCP_IO.Charger[3].inhibited = TRUE AND
	MCP_IO.Charger[4].inhibited = TRUE AND
	MCP_IO.Charger[5].inhibited = TRUE AND
	MCP_IO.Charger[6].inhibited = TRUE
	THEN
		Permissives_DB.AllChargerInhibitON	:= TRUE;
	ELSE
		Permissives_DB.AllChargerInhibitON	:= FALSE;
END_IF;

//add volt fb 1 and 2
IF (ABS(LCP1_IO.Segment[1].Module[1].VoltageFeedback[1]) <= Permissives_DB.CapVoltageThres AND
	ABS(LCP1_IO.Segment[1].Module[1].VoltageFeedback[2]) <= Permissives_DB.CapVoltageThres AND
	ABS(LCP1_IO.Segment[1].Module[2].VoltageFeedback[1]) <= Permissives_DB.CapVoltageThres AND
	ABS(LCP1_IO.Segment[1].Module[2].VoltageFeedback[2]) <= Permissives_DB.CapVoltageThres AND
	ABS(LCP1_IO.Segment[1].Module[3].VoltageFeedback[1]) <= Permissives_DB.CapVoltageThres AND
	ABS(LCP1_IO.Segment[1].Module[3].VoltageFeedback[2]) <= Permissives_DB.CapVoltageThres AND
	ABS(LCP1_IO.Segment[2].Module[4].VoltageFeedback[1]) <= Permissives_DB.CapVoltageThres AND
	ABS(LCP1_IO.Segment[2].Module[4].VoltageFeedback[2]) <= Permissives_DB.CapVoltageThres AND
	ABS(LCP1_IO.Segment[2].Module[5].VoltageFeedback[1]) <= Permissives_DB.CapVoltageThres AND
	ABS(LCP1_IO.Segment[2].Module[5].VoltageFeedback[2]) <= Permissives_DB.CapVoltageThres AND
	ABS(LCP1_IO.Segment[2].Module[6].VoltageFeedback[1]) <= Permissives_DB.CapVoltageThres AND
	ABS(LCP1_IO.Segment[2].Module[6].VoltageFeedback[2]) <= Permissives_DB.CapVoltageThres AND
	ABS(LCP1_IO.Segment[3].Module[7].VoltageFeedback[1]) <= Permissives_DB.CapVoltageThres AND
	ABS(LCP1_IO.Segment[3].Module[7].VoltageFeedback[2]) <= Permissives_DB.CapVoltageThres AND
	ABS(LCP1_IO.Segment[3].Module[8].VoltageFeedback[1]) <= Permissives_DB.CapVoltageThres AND 
	ABS(LCP1_IO.Segment[3].Module[8].VoltageFeedback[2]) <= Permissives_DB.CapVoltageThres AND
	ABS(LCP1_IO.Segment[3].Module[9].VoltageFeedback[1]) <= Permissives_DB.CapVoltageThres AND
	ABS(LCP1_IO.Segment[3].Module[9].VoltageFeedback[2]) <= Permissives_DB.CapVoltageThres AND
	
	ABS(LCP2_IO.Segment[4].Module[1].VoltageFeedback[1]) <= Permissives_DB.CapVoltageThres AND
	ABS(LCP2_IO.Segment[4].Module[1].VoltageFeedback[2]) <= Permissives_DB.CapVoltageThres AND
	ABS(LCP2_IO.Segment[4].Module[2].VoltageFeedback[1]) <= Permissives_DB.CapVoltageThres AND
	ABS(LCP2_IO.Segment[4].Module[2].VoltageFeedback[2]) <= Permissives_DB.CapVoltageThres AND
	ABS(LCP2_IO.Segment[4].Module[3].VoltageFeedback[1]) <= Permissives_DB.CapVoltageThres AND
	ABS(LCP2_IO.Segment[4].Module[3].VoltageFeedback[2]) <= Permissives_DB.CapVoltageThres AND
	ABS(LCP2_IO.Segment[5].Module[4].VoltageFeedback[1]) <= Permissives_DB.CapVoltageThres AND
	ABS(LCP2_IO.Segment[5].Module[4].VoltageFeedback[2]) <= Permissives_DB.CapVoltageThres AND
	ABS(LCP2_IO.Segment[5].Module[5].VoltageFeedback[1]) <= Permissives_DB.CapVoltageThres AND
	ABS(LCP2_IO.Segment[5].Module[5].VoltageFeedback[2]) <= Permissives_DB.CapVoltageThres AND
	ABS(LCP2_IO.Segment[5].Module[6].VoltageFeedback[1]) <= Permissives_DB.CapVoltageThres AND
	ABS(LCP2_IO.Segment[5].Module[6].VoltageFeedback[2]) <= Permissives_DB.CapVoltageThres AND
	ABS(LCP2_IO.Segment[6].Module[7].VoltageFeedback[1]) <= Permissives_DB.CapVoltageThres AND
	ABS(LCP2_IO.Segment[6].Module[7].VoltageFeedback[2]) <= Permissives_DB.CapVoltageThres AND
	ABS(LCP2_IO.Segment[6].Module[8].VoltageFeedback[1]) <= Permissives_DB.CapVoltageThres AND 
	ABS(LCP2_IO.Segment[6].Module[8].VoltageFeedback[2]) <= Permissives_DB.CapVoltageThres AND
	ABS(LCP2_IO.Segment[6].Module[9].VoltageFeedback[1]) <= Permissives_DB.CapVoltageThres AND
	ABS(LCP2_IO.Segment[6].Module[9].VoltageFeedback[2]) <= Permissives_DB.CapVoltageThres) OR HMI_DB.AllCapsDischargedBP = TRUE 
(*  AND all other module voltage feedback <= 40, might need the -ve end & check for valid data*) 
	THEN
		Permissives_DB.AllCapsDischarged := TRUE;
	ELSE 
		Permissives_DB.AllCapsDischarged := FALSE;
END_IF

//VTB status
//LCP1 Voltage Monitor Board bat lo
IF LCP1_IO.VMB.VTB[0].BateryLow = TRUE OR 
	LCP1_IO.VMB.VTB[1].BateryLow = TRUE OR 
	LCP1_IO.VMB.VTB[2].BateryLow = TRUE OR 
	LCP1_IO.VMB.VTB[3].BateryLow = TRUE OR 
	LCP1_IO.VMB.VTB[4].BateryLow = TRUE OR 
	LCP1_IO.VMB.VTB[5].BateryLow = TRUE OR 
	LCP1_IO.VMB.VTB[6].BateryLow = TRUE OR 
	LCP1_IO.VMB.VTB[7].BateryLow = TRUE OR 
	LCP1_IO.VMB.VTB[8].BateryLow = TRUE OR 
	LCP1_IO.VMB.VTB[9].BateryLow = TRUE OR 
	LCP1_IO.VMB.VTB[10].BateryLow = TRUE OR 
	LCP1_IO.VMB.VTB[11].BateryLow = TRUE OR 
	LCP1_IO.VMB.VTB[12].BateryLow = TRUE OR 
	LCP1_IO.VMB.VTB[13].BateryLow = TRUE OR 
	LCP1_IO.VMB.VTB[14].BateryLow = TRUE OR 
	LCP1_IO.VMB.VTB[15].BateryLow = TRUE OR 
	LCP1_IO.VMB.VTB[16].BateryLow = TRUE OR 
	LCP1_IO.VMB.VTB[17].BateryLow = TRUE 
	THEN 
		Permissives_DB.AnyLCP1MonBoardBatLo := TRUE;
	ELSIF 
		LCP1_IO.VMB.VTB[0].BateryLow = FALSE AND 
		LCP1_IO.VMB.VTB[1].BateryLow = FALSE AND 
		LCP1_IO.VMB.VTB[2].BateryLow = FALSE AND 	
		LCP1_IO.VMB.VTB[3].BateryLow = FALSE AND 
		LCP1_IO.VMB.VTB[4].BateryLow = FALSE AND 
		LCP1_IO.VMB.VTB[5].BateryLow = FALSE AND 
		LCP1_IO.VMB.VTB[6].BateryLow = FALSE AND 
		LCP1_IO.VMB.VTB[7].BateryLow = FALSE AND 
		LCP1_IO.VMB.VTB[8].BateryLow = FALSE AND 
		LCP1_IO.VMB.VTB[9].BateryLow = FALSE AND 
		LCP1_IO.VMB.VTB[10].BateryLow = FALSE AND 
		LCP1_IO.VMB.VTB[11].BateryLow = FALSE AND 
		LCP1_IO.VMB.VTB[12].BateryLow = FALSE AND 
		LCP1_IO.VMB.VTB[13].BateryLow = FALSE AND 
		LCP1_IO.VMB.VTB[14].BateryLow = FALSE AND 
		LCP1_IO.VMB.VTB[15].BateryLow = FALSE AND 
		LCP1_IO.VMB.VTB[16].BateryLow = FALSE AND 
		LCP1_IO.VMB.VTB[17].BateryLow = FALSE 
	THEN 
		Permissives_DB.AnyLCP1MonBoardBatLo := FALSE;
END_IF	
//LCP2 Voltage Monitor Board battery lo
IF LCP2_IO.VMB.VTB[0].BateryLow = TRUE OR 
	LCP2_IO.VMB.VTB[1].BateryLow = TRUE OR 
	LCP2_IO.VMB.VTB[2].BateryLow = TRUE OR 
	LCP2_IO.VMB.VTB[3].BateryLow = TRUE OR 
	LCP2_IO.VMB.VTB[4].BateryLow = TRUE OR 
	LCP2_IO.VMB.VTB[5].BateryLow = TRUE OR 
	LCP2_IO.VMB.VTB[6].BateryLow = TRUE OR 
	LCP2_IO.VMB.VTB[7].BateryLow = TRUE OR 
	LCP2_IO.VMB.VTB[8].BateryLow = TRUE OR 
	LCP2_IO.VMB.VTB[9].BateryLow = TRUE OR 
	LCP2_IO.VMB.VTB[10].BateryLow = TRUE OR 
	LCP2_IO.VMB.VTB[11].BateryLow = TRUE OR 
	LCP2_IO.VMB.VTB[12].BateryLow = TRUE OR 
	LCP2_IO.VMB.VTB[13].BateryLow = TRUE OR 
	LCP2_IO.VMB.VTB[14].BateryLow = TRUE OR 
	LCP2_IO.VMB.VTB[15].BateryLow = TRUE OR 
	LCP2_IO.VMB.VTB[16].BateryLow = TRUE OR 
	LCP2_IO.VMB.VTB[17].BateryLow = TRUE 
	THEN 
		Permissives_DB.AnyLCP2MonBoardBatLo := TRUE;
	ELSIF 
		LCP2_IO.VMB.VTB[0].BateryLow = FALSE AND 
		LCP2_IO.VMB.VTB[1].BateryLow = FALSE AND 
		LCP2_IO.VMB.VTB[2].BateryLow = FALSE AND 	
		LCP2_IO.VMB.VTB[3].BateryLow = FALSE AND 
		LCP2_IO.VMB.VTB[4].BateryLow = FALSE AND 
		LCP2_IO.VMB.VTB[5].BateryLow = FALSE AND 
		LCP2_IO.VMB.VTB[6].BateryLow = FALSE AND 
		LCP2_IO.VMB.VTB[7].BateryLow = FALSE AND 
		LCP2_IO.VMB.VTB[8].BateryLow = FALSE AND 
		LCP2_IO.VMB.VTB[9].BateryLow = FALSE AND 
		LCP2_IO.VMB.VTB[10].BateryLow = FALSE AND 
		LCP2_IO.VMB.VTB[11].BateryLow = FALSE AND 
		LCP2_IO.VMB.VTB[12].BateryLow = FALSE AND 
		LCP2_IO.VMB.VTB[13].BateryLow = FALSE AND 
		LCP2_IO.VMB.VTB[14].BateryLow = FALSE AND 
		LCP2_IO.VMB.VTB[15].BateryLow = FALSE AND 
		LCP2_IO.VMB.VTB[16].BateryLow = FALSE AND 
		LCP2_IO.VMB.VTB[17].BateryLow = FALSE 
	THEN 
		Permissives_DB.AnyLCP2MonBoardBatLo := FALSE;
END_IF	
//lcp1 volt montiro board loss HB
IF LCP1_IO.VMB.VTB[0].LossVoltTransBoard = TRUE OR 
	LCP1_IO.VMB.VTB[1].LossVoltTransBoard = TRUE OR 
	LCP1_IO.VMB.VTB[2].LossVoltTransBoard = TRUE OR 
	LCP1_IO.VMB.VTB[3].LossVoltTransBoard = TRUE OR 
	LCP1_IO.VMB.VTB[4].LossVoltTransBoard = TRUE OR 
	LCP1_IO.VMB.VTB[5].LossVoltTransBoard = TRUE OR 
	LCP1_IO.VMB.VTB[6].LossVoltTransBoard = TRUE OR 
	LCP1_IO.VMB.VTB[7].LossVoltTransBoard = TRUE OR 
	LCP1_IO.VMB.VTB[8].LossVoltTransBoard = TRUE OR 
	LCP1_IO.VMB.VTB[9].LossVoltTransBoard = TRUE OR 
	LCP1_IO.VMB.VTB[10].LossVoltTransBoard = TRUE OR 
	LCP1_IO.VMB.VTB[11].LossVoltTransBoard = TRUE OR 
	LCP1_IO.VMB.VTB[12].LossVoltTransBoard = TRUE OR 
	LCP1_IO.VMB.VTB[13].LossVoltTransBoard = TRUE OR 
	LCP1_IO.VMB.VTB[14].LossVoltTransBoard = TRUE OR 
	LCP1_IO.VMB.VTB[15].LossVoltTransBoard = TRUE OR 
	LCP1_IO.VMB.VTB[16].LossVoltTransBoard = TRUE OR 
	LCP1_IO.VMB.VTB[17].LossVoltTransBoard = TRUE 
	THEN 
		Permissives_DB.AnyLCP1MonBoardLoss := TRUE;
	ELSIF 
		LCP1_IO.VMB.VTB[0].LossVoltTransBoard = FALSE AND 
		LCP1_IO.VMB.VTB[1].LossVoltTransBoard = FALSE AND 
		LCP1_IO.VMB.VTB[2].LossVoltTransBoard = FALSE AND 	
		LCP1_IO.VMB.VTB[3].LossVoltTransBoard = FALSE AND 
		LCP1_IO.VMB.VTB[4].LossVoltTransBoard = FALSE AND 
		LCP1_IO.VMB.VTB[5].LossVoltTransBoard = FALSE AND 
		LCP1_IO.VMB.VTB[6].LossVoltTransBoard = FALSE AND 
		LCP1_IO.VMB.VTB[7].LossVoltTransBoard = FALSE AND 
		LCP1_IO.VMB.VTB[8].LossVoltTransBoard = FALSE AND 
		LCP1_IO.VMB.VTB[9].LossVoltTransBoard = FALSE AND 
		LCP1_IO.VMB.VTB[10].LossVoltTransBoard = FALSE AND 
		LCP1_IO.VMB.VTB[11].LossVoltTransBoard = FALSE AND 
		LCP1_IO.VMB.VTB[12].LossVoltTransBoard = FALSE AND 
		LCP1_IO.VMB.VTB[13].LossVoltTransBoard = FALSE AND 
		LCP1_IO.VMB.VTB[14].LossVoltTransBoard = FALSE AND 
		LCP1_IO.VMB.VTB[15].LossVoltTransBoard = FALSE AND 
		LCP1_IO.VMB.VTB[16].LossVoltTransBoard = FALSE AND 
		LCP1_IO.VMB.VTB[17].LossVoltTransBoard = FALSE 
	THEN 
		Permissives_DB.AnyLCP1MonBoardLoss := FALSE;
END_IF 
//lcp2 volt montiro board loss HB
IF LCP2_IO.VMB.VTB[0].LossVoltTransBoard = TRUE OR 
	LCP2_IO.VMB.VTB[1].LossVoltTransBoard = TRUE OR 
	LCP2_IO.VMB.VTB[2].LossVoltTransBoard = TRUE OR 
	LCP2_IO.VMB.VTB[3].LossVoltTransBoard = TRUE OR 
	LCP2_IO.VMB.VTB[4].LossVoltTransBoard = TRUE OR 
	LCP2_IO.VMB.VTB[5].LossVoltTransBoard = TRUE OR 
	LCP2_IO.VMB.VTB[6].LossVoltTransBoard = TRUE OR 
	LCP2_IO.VMB.VTB[7].LossVoltTransBoard = TRUE OR 
	LCP2_IO.VMB.VTB[8].LossVoltTransBoard = TRUE OR 
	LCP2_IO.VMB.VTB[9].LossVoltTransBoard = TRUE OR 
	LCP2_IO.VMB.VTB[10].LossVoltTransBoard = TRUE OR 
	LCP2_IO.VMB.VTB[11].LossVoltTransBoard = TRUE OR 
	LCP2_IO.VMB.VTB[12].LossVoltTransBoard = TRUE OR 
	LCP2_IO.VMB.VTB[13].LossVoltTransBoard = TRUE OR 
	LCP2_IO.VMB.VTB[14].LossVoltTransBoard = TRUE OR 
	LCP2_IO.VMB.VTB[15].LossVoltTransBoard = TRUE OR 
	LCP2_IO.VMB.VTB[16].LossVoltTransBoard = TRUE OR 
	LCP2_IO.VMB.VTB[17].LossVoltTransBoard = TRUE 
	THEN 
		Permissives_DB.AnyLCP2MonBoardLoss := TRUE;
	ELSIF 
		LCP2_IO.VMB.VTB[0].LossVoltTransBoard = FALSE AND 
		LCP2_IO.VMB.VTB[1].LossVoltTransBoard = FALSE AND 
		LCP2_IO.VMB.VTB[2].LossVoltTransBoard = FALSE AND 	
		LCP2_IO.VMB.VTB[3].LossVoltTransBoard = FALSE AND 
		LCP2_IO.VMB.VTB[4].LossVoltTransBoard = FALSE AND 
		LCP2_IO.VMB.VTB[5].LossVoltTransBoard = FALSE AND 
		LCP2_IO.VMB.VTB[6].LossVoltTransBoard = FALSE AND 
		LCP2_IO.VMB.VTB[7].LossVoltTransBoard = FALSE AND 
		LCP2_IO.VMB.VTB[8].LossVoltTransBoard = FALSE AND 
		LCP2_IO.VMB.VTB[9].LossVoltTransBoard = FALSE AND 
		LCP2_IO.VMB.VTB[10].LossVoltTransBoard = FALSE AND 
		LCP2_IO.VMB.VTB[11].LossVoltTransBoard = FALSE AND 
		LCP2_IO.VMB.VTB[12].LossVoltTransBoard = FALSE AND 
		LCP2_IO.VMB.VTB[13].LossVoltTransBoard = FALSE AND 
		LCP2_IO.VMB.VTB[14].LossVoltTransBoard = FALSE AND 
		LCP2_IO.VMB.VTB[15].LossVoltTransBoard = FALSE AND 
		LCP2_IO.VMB.VTB[16].LossVoltTransBoard = FALSE AND 
		LCP2_IO.VMB.VTB[17].LossVoltTransBoard = FALSE 
	THEN 
		Permissives_DB.AnyLCP2MonBoardLoss := FALSE;
END_IF 

IF Permissives_DB.AnyLCP1MonBoardBatLo = TRUE OR Permissives_DB.AnyLCP2MonBoardBatLo = TRUE 
	THEN 
		Permissives_DB.AnyVoltMonBoardBatLo := TRUE;
	ELSIF 
		Permissives_DB.AnyLCP1MonBoardBatLo = FALSE AND Permissives_DB.AnyLCP2MonBoardBatLo = FALSE 
	THEN 
		Permissives_DB.AnyVoltMonBoardBatLo := FALSE;
END_IF

IF Permissives_DB.AnyLCP1MonBoardLoss = TRUE OR Permissives_DB.AnyLCP2MonBoardLoss = TRUE 
	THEN 
		Permissives_DB.AnyVoltMonBoardLoss := TRUE;
	ELSIF 
		Permissives_DB.AnyLCP1MonBoardLoss = FALSE AND Permissives_DB.AnyLCP2MonBoardLoss = FALSE 
	THEN 
		Permissives_DB.AnyVoltMonBoardLoss := FALSE;
END_IF

IF (Permissives_DB.ChargerVBelowThres = TRUE AND 
	Permissives_DB.AllChargerHVisOFF = TRUE AND 
	//Permissives_DB.AllChargerInhibitON	= TRUE AND 
	Permissives_DB.AllDumpRelayOpen = FALSE AND 
	Permissives_DB.AllCapsDischarged = TRUE) OR HMI_DB.SystemSafeBP = TRUE 
THEN
	(*MCP_IO.Charger[2].voltageFeedback <= 10 AND *)
	Permissives_DB.SystemIsSafe := TRUE;
	ELSE
		Permissives_DB.SystemIsSafe := FALSE;
END_IF
		
IF Permissives_DB.AllCapsDischarged = TRUE THEN 
	LCP1_IO.SegmentCharged := FALSE; //for status light only
	LCP2_IO.SegmentCharged := FALSE; //for status light only
END_IF

IF MCP_IO.Charger[1].EndOfCharge = TRUE AND
	MCP_IO.Charger[2].EndOfCharge = TRUE AND
	MCP_IO.Charger[3].EndOfCharge = TRUE AND
	MCP_IO.Charger[4].EndOfCharge = TRUE AND
	MCP_IO.Charger[5].EndOfCharge = TRUE AND
	MCP_IO.Charger[6].EndOfCharge = TRUE 
THEN
	Permissives_DB.AllChargerEOC := TRUE;
	ELSE
		Permissives_DB.AllChargerEOC := FALSE;
END_IF;

// might or might not beused for the seq
IF MCP_IO.PSU1_DCOK = TRUE AND LCP1_IO.PSU1OK = TRUE AND LCP2_IO.PSU1OK = TRUE THEN
	Trips_DB.AllDCpsuOK := TRUE;
	ELSE
		Trips_DB.AllDCpsuOK := FALSE;
END_IF

IF MCP_IO.MasterStopPB_NotPressed = FALSE THEN 
	Trips_DB.MasterSTOPPressed := TRUE;
	ELSE
		Trips_DB.MasterSTOPPressed := FALSE;
END_IF

IF MCP_IO.CageEstopCircuitOK = FALSE OR MCP_IO.MasterStopPB_NotPressed = FALSE THEN 
	Trips_DB.AnyEstopPressed := TRUE;
END_IF

END_PROGRAM

// ---- POUs/AnalogConversion.TcPOU
PROGRAM AnalogConversion
VAR
	i					: INT := 1; //charger 1-6
	j					: INT := 1;  // section 1 - 4 
	k					: INT := 1;  // cap 1-10
	m					: INT := 1; //form cap 1-12
	n					: INT := 7;
	VoltMonAC1			: ARRAY[1..18] OF VoltMonAC_FB;
	VoltMonAC2			: ARRAY[1..18] OF VoltMonAC_FB;
END_VAR

//MCP Charger 
//Analog Input
FOR i := 1 TO n BY 1 DO 
	//MCP_IO.Charger[i].voltageSP := (HMI_DB.TDKLoad[i].RequiredChargedV *1000);
	MCP_IO.Charger[i].voltageSP := (1000*Setpoints.TDKLoad[i].RequiredChargedV);
END_FOR

//AI
FOR i := 1 TO n BY 1 DO
	//voltage
	MCP_IO.Charger[i].voltageFeedback_norm := Norm_x (raw_input := INT_TO_REAL (MCP_IO.Charger[i].voltageFeedback_raw),
														x_max := 32767,
														x_min := 0);
	//current																									
	MCP_IO.Charger[i].currentFeedback_norm := Norm_x (raw_input := INT_TO_REAL (MCP_IO.Charger[i].currentFeedback_raw),
														x_max := 32767,
														x_min := 0);
	//50kV chargers feedback
	//if 50kV config selected
	IF MCP_IO.Charger[i].ChargerType = E_ChargerType.TDK50kV THEN 
		//50kv
		MCP_IO.Charger[i].voltageFeedback := (EngVal.Max_50kVChargerVoltage - EngVal.Min_50kVChargerVoltage) * ADC_10V(
																							normal_input := MCP_IO.Charger[i].voltageFeedback_norm,
																							x_max := 10,
																							x_min := 0);

		MCP_IO.Charger[i].currentFeedback := (EngVal.Max_50kVChargerCurrent - EngVal.Min_50kVChargerCurrent) * ADC_10V(
																							normal_input := MCP_IO.Charger[i].currentFeedback_norm,
																							x_max := 10,
																							x_min := 0);
		//12kv
	ELSIF MCP_IO.Charger[i].ChargerType = E_ChargerType.TDK12kV THEN
		MCP_IO.Charger[i].voltageFeedback := (EngVal.Max_12kVChargerVoltage - EngVal.Min_12kVChargerVoltage) * ADC_10V(
																							normal_input := MCP_IO.Charger[i].voltageFeedback_norm,
																							x_max := 10,
																							x_min := 0);
		MCP_IO.Charger[i].currentFeedback := (EngVal.Max_12kVChargerCurrent - EngVal.Min_12kVChargerCurrent) * ADC_10V(
																							normal_input := MCP_IO.Charger[i].currentFeedback_norm,
																							x_max := 10,
																							x_min := 0);	
	ELSIF MCP_IO.Charger[i].ChargerType = E_ChargerType.TDK30kV THEN
		MCP_IO.Charger[i].voltageFeedback := (EngVal.Max_30kVChargerVoltage - EngVal.Min_30kVChargerVoltage) * ADC_10V(
																							normal_input := MCP_IO.Charger[i].voltageFeedback_norm,
																							x_max := 10,
																							x_min := 0);														
		// 30kV charger max current output is 0.6A													
		MCP_IO.Charger[i].currentFeedback := (EngVal.Max_30kVChargerCurrent - EngVal.Min_30kVChargerCurrent) * ADC_10V(
																							normal_input := MCP_IO.Charger[i].currentFeedback_norm,
																							x_max := 10,
																							x_min := 0);							
	END_IF;	
END_FOR;

//Analog Output
//voltageSP = Required Charge Voltage******************
//limit for charing the cap
//FOR i := 1 TO 8 BY 1 DO
FOR i := 1 TO n BY 1 DO	
	
	//if 50kV config selected
	IF MCP_IO.Charger[i].ChargerType = E_ChargerType.TDK50kV THEN 
		//set limits of charger voltage input 
		IF MCP_IO.Charger[i].voltageSP >= (EngVal.UpperLimit50kVCaps) THEN
			MCP_IO.Charger[i].voltageSP := 35000; //limit at 35kV
		ELSIF MCP_IO.Charger[i].voltageSP <= 0 THEN
			MCP_IO.Charger[i].voltageSP := 0; //limit at 0V
		END_IF; 
		
		//prepare output signal for 50kV chargers.
		MCP_IO.Charger[i].voltageSP_norm := Norm_x (raw_input :=(MCP_IO.Charger[i].voltageSP), 
												x_max := EngVal.Max_50kVChargerVoltage,
												x_min := EngVal.Min_50kVChargerVoltage);	
												
		MCP_IO.Charger[i].voltageSP_raw := AQ (norm_input := MCP_IO.Charger[i].voltageSP_norm, 
												x_max := 10,
												x_min := 0);
												
	ELSIF MCP_IO.Charger[i].ChargerType = E_ChargerType.TDK12kV THEN 
		//set limits of charger voltage input 
		IF MCP_IO.Charger[i].voltageSP >= (EngVal.UpperLimit12kVCaps) THEN
			MCP_IO.Charger[i].voltageSP := 10500; //limit at 35kV
		ELSIF MCP_IO.Charger[i].voltageSP <= 0 THEN
			MCP_IO.Charger[i].voltageSP := ABS(MCP_IO.Charger[i].voltageSP); //limit at 0V
		END_IF; 
		
		//prepare output signal for 50kV chargers.
		MCP_IO.Charger[i].voltageSP_norm := Norm_x (raw_input :=(MCP_IO.Charger[i].voltageSP), 
												x_max := EngVal.Max_12kVChargerVoltage,
												x_min := EngVal.Min_12kVChargerVoltage);	
												
		MCP_IO.Charger[i].voltageSP_raw := AQ (norm_input := MCP_IO.Charger[i].voltageSP_norm, 
												x_max := 10,
												x_min := 0);
	
	ELSIF MCP_IO.Charger[i].ChargerType = E_ChargerType.TDK30kV THEN 		
		//set limits of charger voltage input 
		IF MCP_IO.Charger[i].voltageSP >= (EngVal.UpperLimit12kVCaps) THEN
			MCP_IO.Charger[i].voltageSP := 10500; //limit at 35kV
		ELSIF MCP_IO.Charger[i].voltageSP <= 0 THEN
			MCP_IO.Charger[i].voltageSP := ABS(MCP_IO.Charger[i].voltageSP); //limit at 0V
		END_IF;
		//prepare output signal for 30kV chargers.
		MCP_IO.Charger[i].voltageSP_norm := Norm_x (raw_input :=(MCP_IO.Charger[i].voltageSP), 
												x_max := EngVal.Max_30kVChargerVoltage,
												x_min := EngVal.Min_30kVChargerVoltage);	
												
		MCP_IO.Charger[i].voltageSP_raw := AQ (norm_input := MCP_IO.Charger[i].voltageSP_norm, 
												x_max := 10,
												x_min := 0);
	END_IF;	
												
	//limite for output sigal (<= 10V)  this should not happen
	IF MCP_IO.Charger[i].voltageSP_raw >= 32767 THEN 
		MCP_IO.Charger[i].voltageSP_raw := 32767; 										
	END_IF;
	
END_FOR;

//Cap voltage feedback
(*
//can also add a range of x samples for self calibrating **note: normalized range needs to be calibrated for each board
VoltMonitor_DB.VoltageReading_norm[0] := Norm_x (raw_input := INT_TO_REAL (VoltMonitor_DB.VoltageReading_raw[0]),
													x_max := 904, //10bit value - 1110001000 = 904deci
													x_min := 100); //100deci is the zero of range -1.61 to 12.01
LCP1_IO.Segment[1].Module[1].VoltageFeedback[1] := (12010 - 0) * ADC_10V(normal_input := VoltMonitor_DB.VoltageReading_norm[0],
																		x_max := 12.01,
																		x_min := 0); //use zero, it will cal for the -ve	

*)

(* // changed to a FB for norm and ADC
LCP1_IO.Segment[1].Module[1].VoltageFeedback_norm[1] := Norm_x (raw_input := INT_TO_REAL (LCP1_IO.Segment[1].Module[1].VoltageFeedback_raw[1]),
													x_max := 904, //10bit value - 1110001000 = 904deci
													x_min := 100); //100deci is the zero of range -1.61 to 12.01
LCP1_IO.Segment[1].Module[1].VoltageFeedback[1] := (12010 - 0) * ADC_10V(normal_input := LCP1_IO.Segment[1].Module[1].VoltageFeedback_norm[1],
																		x_max := 12.01,
																		x_min := 0); //use zero, it will cal for the -ve
*)
// using FB instead.
VoltMonAC1[1](raw_input := DINT_TO_REAL(LCP1_IO.Segment[1].Module[1].VoltageFeedback_raw[1]),
				norm_x_max := 904, //individually calibrated, otherwise can do a for loop
				norm_x_min := 100, 
				RangUpp := 12.01, 
				RangLow := 0, 
				ADC_max := 12010, 
				ADC_min := 0, 
				voltage_reading => LCP1_IO.Segment[1].Module[1].VoltageFeedback[1]);

VoltMonAC1[2](raw_input := DINT_TO_REAL(LCP1_IO.Segment[1].Module[1].VoltageFeedback_raw[2]),
				norm_x_max := 904, 
				norm_x_min := 100, 
				RangUpp := 12.01, 
				RangLow := 0, 
				ADC_max := 12010, 
				ADC_min := 0, 
				voltage_reading => LCP1_IO.Segment[1].Module[1].VoltageFeedback[2]);		

VoltMonAC1[3](raw_input := DINT_TO_REAL(LCP1_IO.Segment[1].Module[2].VoltageFeedback_raw[1]),
				norm_x_max := 904, 
				norm_x_min := 100, 
				RangUpp := 12.01, 
				RangLow := 0, 
				ADC_max := 12010, 
				ADC_min := 0, 
				voltage_reading => LCP1_IO.Segment[1].Module[2].VoltageFeedback[1]);	
				
VoltMonAC1[4](raw_input := DINT_TO_REAL(LCP1_IO.Segment[1].Module[2].VoltageFeedback_raw[2]),
				norm_x_max := 904, 
				norm_x_min := 100, 
				RangUpp := 12.01, 
				RangLow := 0, 
				ADC_max := 12010, 
				ADC_min := 0, 
				voltage_reading => LCP1_IO.Segment[1].Module[2].VoltageFeedback[2]);					

VoltMonAC1[5](raw_input := DINT_TO_REAL(LCP1_IO.Segment[1].Module[3].VoltageFeedback_raw[1]),
				norm_x_max := 904, 
				norm_x_min := 100, 
				RangUpp := 12.01, 
				RangLow := 0, 
				ADC_max := 12010, 
				ADC_min := 0, 
				voltage_reading => LCP1_IO.Segment[1].Module[3].VoltageFeedback[1]);	
				
VoltMonAC1[6](raw_input := DINT_TO_REAL(LCP1_IO.Segment[1].Module[3].VoltageFeedback_raw[2]),
				norm_x_max := 904, 
				norm_x_min := 100, 
				RangUpp := 12.01, 
				RangLow := 0, 
				ADC_max := 12010, 
				ADC_min := 0, 
				voltage_reading => LCP1_IO.Segment[1].Module[3].VoltageFeedback[2]);				
				
VoltMonAC1[7](raw_input := DINT_TO_REAL(LCP1_IO.Segment[2].Module[4].VoltageFeedback_raw[1]),
				norm_x_max := 904, 
				norm_x_min := 100, 
				RangUpp := 12.01, 
				RangLow := 0, 
				ADC_max := 12010, 
				ADC_min := 0, 
				voltage_reading => LCP1_IO.Segment[2].Module[4].VoltageFeedback[1]);	
				
VoltMonAC1[8](raw_input := DINT_TO_REAL(LCP1_IO.Segment[2].Module[4].VoltageFeedback_raw[2]),
				norm_x_max := 904, 
				norm_x_min := 100, 
				RangUpp := 12.01, 
				RangLow := 0, 
				ADC_max := 12010, 
				ADC_min := 0, 
				voltage_reading => LCP1_IO.Segment[2].Module[4].VoltageFeedback[2]);
	
VoltMonAC1[9](raw_input := DINT_TO_REAL(LCP1_IO.Segment[2].Module[5].VoltageFeedback_raw[1]),
				norm_x_max := 904, 
				norm_x_min := 100, 
				RangUpp := 12.01, 
				RangLow := 0, 
				ADC_max := 12010, 
				ADC_min := 0, 
				voltage_reading => LCP1_IO.Segment[2].Module[5].VoltageFeedback[1]);	
				
VoltMonAC1[10](raw_input := DINT_TO_REAL(LCP1_IO.Segment[2].Module[5].VoltageFeedback_raw[2]),
				norm_x_max := 904, 
				norm_x_min := 100, 
				RangUpp := 12.01, 
				RangLow := 0, 
				ADC_max := 12010, 
				ADC_min := 0, 
				voltage_reading => LCP1_IO.Segment[2].Module[5].VoltageFeedback[2]);
				
VoltMonAC1[11](raw_input := DINT_TO_REAL(LCP1_IO.Segment[2].Module[6].VoltageFeedback_raw[1]),
				norm_x_max := 904, 
				norm_x_min := 100, 
				RangUpp := 12.01, 
				RangLow := 0, 
				ADC_max := 12010, 
				ADC_min := 0, 
				voltage_reading => LCP1_IO.Segment[2].Module[6].VoltageFeedback[1]);	
				
VoltMonAC1[12](raw_input := DINT_TO_REAL(LCP1_IO.Segment[2].Module[6].VoltageFeedback_raw[2]),
				norm_x_max := 904, 
				norm_x_min := 100, 
				RangUpp := 12.01, 
				RangLow := 0, 
				ADC_max := 12010, 
				ADC_min := 0, 
				voltage_reading => LCP1_IO.Segment[2].Module[6].VoltageFeedback[2]);			

VoltMonAC1[13](raw_input := DINT_TO_REAL(LCP1_IO.Segment[3].Module[7].VoltageFeedback_raw[1]),
				norm_x_max := 904, 
				norm_x_min := 100, 
				RangUpp := 12.01, 
				RangLow := 0, 
				ADC_max := 12010, 
				ADC_min := 0, 
				voltage_reading => LCP1_IO.Segment[3].Module[7].VoltageFeedback[1]);	
				
VoltMonAC1[14](raw_input := DINT_TO_REAL(LCP1_IO.Segment[3].Module[7].VoltageFeedback_raw[2]),
				norm_x_max := 904, 
				norm_x_min := 100, 
				RangUpp := 12.01, 
				RangLow := 0, 
				ADC_max := 12010, 
				ADC_min := 0, 
				voltage_reading => LCP1_IO.Segment[3].Module[7].VoltageFeedback[2]);
				
VoltMonAC1[15](raw_input := DINT_TO_REAL(LCP1_IO.Segment[3].Module[8].VoltageFeedback_raw[1]),
				norm_x_max := 904, 
				norm_x_min := 100, 
				RangUpp := 12.01, 
				RangLow := 0, 
				ADC_max := 12010, 
				ADC_min := 0, 
				voltage_reading => LCP1_IO.Segment[3].Module[8].VoltageFeedback[1]);	
				
VoltMonAC1[16](raw_input := DINT_TO_REAL(LCP1_IO.Segment[3].Module[8].VoltageFeedback_raw[2]),
				norm_x_max := 904, 
				norm_x_min := 100, 
				RangUpp := 12.01, 
				RangLow := 0, 
				ADC_max := 12010, 
				ADC_min := 0, 
				voltage_reading => LCP1_IO.Segment[3].Module[8].VoltageFeedback[2]);
				
VoltMonAC1[17](raw_input := DINT_TO_REAL(LCP1_IO.Segment[3].Module[9].VoltageFeedback_raw[1]),
				norm_x_max := 904, 
				norm_x_min := 100, 
				RangUpp := 12.01, 
				RangLow := 0, 
				ADC_max := 12010, 
				ADC_min := 0, 
				voltage_reading => LCP1_IO.Segment[3].Module[9].VoltageFeedback[1]);	
				
VoltMonAC1[18](raw_input := DINT_TO_REAL(LCP1_IO.Segment[3].Module[9].VoltageFeedback_raw[2]),
				norm_x_max := 904, 
				norm_x_min := 100, 
				RangUpp := 12.01, 
				RangLow := 0, 
				ADC_max := 12010, 
				ADC_min := 0, 
				voltage_reading => LCP1_IO.Segment[3].Module[9].VoltageFeedback[2]);	

//lcp2 cap voltage mon adc
VoltMonAC2[1](raw_input := DINT_TO_REAL(LCP2_IO.Segment[4].Module[1].VoltageFeedback_raw[1]),
				norm_x_max := 904, //individually calibrated, otherwise can do a for loop
				norm_x_min := 100, 
				RangUpp := 12.01, 
				RangLow := 0, 
				ADC_max := 12010, 
				ADC_min := 0, 
				voltage_reading => LCP2_IO.Segment[4].Module[1].VoltageFeedback[1]);

VoltMonAC2[2](raw_input := DINT_TO_REAL(LCP2_IO.Segment[4].Module[1].VoltageFeedback_raw[2]),
				norm_x_max := 904, 
				norm_x_min := 100, 
				RangUpp := 12.01, 
				RangLow := 0, 
				ADC_max := 12010, 
				ADC_min := 0, 
				voltage_reading => LCP2_IO.Segment[4].Module[1].VoltageFeedback[2]);		

VoltMonAC2[3](raw_input := DINT_TO_REAL(LCP2_IO.Segment[4].Module[2].VoltageFeedback_raw[1]),
				norm_x_max := 904, 
				norm_x_min := 100, 
				RangUpp := 12.01, 
				RangLow := 0, 
				ADC_max := 12010, 
				ADC_min := 0, 
				voltage_reading => LCP2_IO.Segment[4].Module[2].VoltageFeedback[1]);	
				
VoltMonAC2[4](raw_input := DINT_TO_REAL(LCP2_IO.Segment[4].Module[2].VoltageFeedback_raw[2]),
				norm_x_max := 904, 
				norm_x_min := 100, 
				RangUpp := 12.01, 
				RangLow := 0, 
				ADC_max := 12010, 
				ADC_min := 0, 
				voltage_reading => LCP2_IO.Segment[4].Module[2].VoltageFeedback[2]);					

VoltMonAC2[5](raw_input := DINT_TO_REAL(LCP2_IO.Segment[4].Module[3].VoltageFeedback_raw[1]),
				norm_x_max := 904, 
				norm_x_min := 100, 
				RangUpp := 12.01, 
				RangLow := 0, 
				ADC_max := 12010, 
				ADC_min := 0, 
				voltage_reading => LCP2_IO.Segment[4].Module[3].VoltageFeedback[1]);	
				
VoltMonAC2[6](raw_input := DINT_TO_REAL(LCP2_IO.Segment[4].Module[3].VoltageFeedback_raw[2]),
				norm_x_max := 904, 
				norm_x_min := 100, 
				RangUpp := 12.01, 
				RangLow := 0, 
				ADC_max := 12010, 
				ADC_min := 0, 
				voltage_reading => LCP2_IO.Segment[4].Module[3].VoltageFeedback[2]);				
				
VoltMonAC2[7](raw_input := DINT_TO_REAL(LCP2_IO.Segment[5].Module[4].VoltageFeedback_raw[1]),
				norm_x_max := 904, 
				norm_x_min := 100, 
				RangUpp := 12.01, 
				RangLow := 0, 
				ADC_max := 12010, 
				ADC_min := 0, 
				voltage_reading => LCP2_IO.Segment[5].Module[4].VoltageFeedback[1]);	
				
VoltMonAC2[8](raw_input := DINT_TO_REAL(LCP2_IO.Segment[5].Module[4].VoltageFeedback_raw[2]),
				norm_x_max := 904, 
				norm_x_min := 100, 
				RangUpp := 12.01, 
				RangLow := 0, 
				ADC_max := 12010, 
				ADC_min := 0, 
				voltage_reading => LCP2_IO.Segment[5].Module[4].VoltageFeedback[2]);
	
VoltMonAC2[9](raw_input := DINT_TO_REAL(LCP2_IO.Segment[5].Module[5].VoltageFeedback_raw[1]),
				norm_x_max := 904, 
				norm_x_min := 100, 
				RangUpp := 12.01, 
				RangLow := 0, 
				ADC_max := 12010, 
				ADC_min := 0, 
				voltage_reading => LCP2_IO.Segment[5].Module[5].VoltageFeedback[1]);	
				
VoltMonAC2[10](raw_input := DINT_TO_REAL(LCP2_IO.Segment[5].Module[5].VoltageFeedback_raw[2]),
				norm_x_max := 904, 
				norm_x_min := 100, 
				RangUpp := 12.01, 
				RangLow := 0, 
				ADC_max := 12010, 
				ADC_min := 0, 
				voltage_reading => LCP2_IO.Segment[5].Module[5].VoltageFeedback[2]);
				
VoltMonAC2[11](raw_input := DINT_TO_REAL(LCP2_IO.Segment[5].Module[6].VoltageFeedback_raw[1]),
				norm_x_max := 904, 
				norm_x_min := 100, 
				RangUpp := 12.01, 
				RangLow := 0, 
				ADC_max := 12010, 
				ADC_min := 0, 
				voltage_reading => LCP2_IO.Segment[5].Module[6].VoltageFeedback[1]);	
				
VoltMonAC2[12](raw_input := DINT_TO_REAL(LCP2_IO.Segment[5].Module[6].VoltageFeedback_raw[2]),
				norm_x_max := 904, 
				norm_x_min := 100, 
				RangUpp := 12.01, 
				RangLow := 0, 
				ADC_max := 12010, 
				ADC_min := 0, 
				voltage_reading => LCP2_IO.Segment[5].Module[6].VoltageFeedback[2]);			

VoltMonAC2[13](raw_input := DINT_TO_REAL(LCP2_IO.Segment[6].Module[7].VoltageFeedback_raw[1]),
				norm_x_max := 904, 
				norm_x_min := 100, 
				RangUpp := 12.01, 
				RangLow := 0, 
				ADC_max := 12010, 
				ADC_min := 0, 
				voltage_reading => LCP2_IO.Segment[6].Module[7].VoltageFeedback[1]);	
				
VoltMonAC2[14](raw_input := DINT_TO_REAL(LCP2_IO.Segment[6].Module[7].VoltageFeedback_raw[2]),
				norm_x_max := 904, 
				norm_x_min := 100, 
				RangUpp := 12.01, 
				RangLow := 0, 
				ADC_max := 12010, 
				ADC_min := 0, 
				voltage_reading => LCP2_IO.Segment[6].Module[7].VoltageFeedback[2]);
				
VoltMonAC2[15](raw_input := DINT_TO_REAL(LCP2_IO.Segment[6].Module[8].VoltageFeedback_raw[1]),
				norm_x_max := 904, 
				norm_x_min := 100, 
				RangUpp := 12.01, 
				RangLow := 0, 
				ADC_max := 12010, 
				ADC_min := 0, 
				voltage_reading => LCP2_IO.Segment[6].Module[8].VoltageFeedback[1]);	
				
VoltMonAC2[16](raw_input := DINT_TO_REAL(LCP2_IO.Segment[6].Module[8].VoltageFeedback_raw[2]),
				norm_x_max := 904, 
				norm_x_min := 100, 
				RangUpp := 12.01, 
				RangLow := 0, 
				ADC_max := 12010, 
				ADC_min := 0, 
				voltage_reading => LCP2_IO.Segment[6].Module[8].VoltageFeedback[2]);
				
VoltMonAC2[17](raw_input := DINT_TO_REAL(LCP2_IO.Segment[6].Module[9].VoltageFeedback_raw[1]),
				norm_x_max := 904, 
				norm_x_min := 100, 
				RangUpp := 12.01, 
				RangLow := 0, 
				ADC_max := 12010, 
				ADC_min := 0, 
				voltage_reading => LCP2_IO.Segment[6].Module[9].VoltageFeedback[1]);	
				
VoltMonAC2[18](raw_input := DINT_TO_REAL(LCP2_IO.Segment[6].Module[9].VoltageFeedback_raw[2]),
				norm_x_max := 904, 
				norm_x_min := 100, 
				RangUpp := 12.01, 
				RangLow := 0, 
				ADC_max := 12010, 
				ADC_min := 0, 
				voltage_reading => LCP2_IO.Segment[6].Module[9].VoltageFeedback[2]);	
					
//reset counter
//IF i > 8 THEN
IF i > n THEN
	i := 1;
END_IF;

IF j > 3 THEN 
	j := 1;
END_IF

IF k > 10 THEN 
	k := 1;
END_IF

IF m > 12 THEN 
	m := 1;
END_IF

END_PROGRAM

// ---- POUs/VoltMonAC_FB.TcPOU
FUNCTION_BLOCK VoltMonAC_FB
VAR_INPUT
	raw_input : REAL;
	norm_x_max : REAL := 10;
	norm_x_min : REAL := 0;
	RangUpp : REAL := 12.1;
	RangLow : REAL := 0;
	ADC_max : REAL := 12100;
	ADC_min	: REAL := 0;
END_VAR
VAR_OUTPUT
	voltage_reading : REAL;
END_VAR
VAR
	normal_input : REAL;
END_VAR

normal_input := Norm_x (raw_input := raw_input,
						x_max := norm_x_max, //10bit value - 1110001000 = 904deci
						x_min := norm_x_min); //100deci is the zero of range -1.61 to 12.01
voltage_reading := (ADC_max - ADC_min) * ADC_10V(normal_input := normal_input,
													x_max := RangUpp,
													x_min := RangLow); //use zero, it will cal for the -ve

END_FUNCTION_BLOCK

// ---- POUs/VoltageMonitor.TcPOU
PROGRAM VoltageMonitor
VAR
	i : USINT := 1;
	j : INT := 1;
	k : USINT := 0;
	eVoltFB : E_VoltFB;
	
	m : USINT := 0; //0-18
	n : INT := 0; //
	p : INT := -3;
	q : INT := 3;

	counter : USINT := 0;
	b : ARRAY[0..3] OF BOOL;
	b1 : BOOL;
	b2 : BOOL;
	b3 : BOOL;
	//pause : BOOL;
	//VMBoardWDT_TON : ARRAY[0..24] OF TON;
	//VMBoardWDT_PT	: TIME := T#2S;
	//VMBoardWDT_ET	: TIME;
	//DataNull	: ARRAY[0..24] OF BOOL ;
	//DataNullRebunceTMR_TON : ARRAY[0..24] OF TON;
	//DataNullRebounce_PT	: TIME := T#800MS;
	//DataNullRebounce	: ARRAY[0..24] OF BOOL ;
	VMB1 : ARRAY[0..17] OF VoltTranBd;
	VMB2 : ARRAY[0..17] OF VoltTranBd;
END_VAR

//2 voltage tran borad per module, total of 36 channels for M1 
//volt monitor board 1 - trans board 0
FOR m := 0 TO 17 BY 1 DO 
	VMB1[m] ( CapRaw := LCP1_IO.VMB.VTB[m].CapRaw );		
	LCP1_IO.VMB.VTB[m].BateryLow 						:= VMB1[m].BatteryLow;
	LCP1_IO.VMB.VTB[m].VoltageReading_raw				:= VMB1[m].VoltageReading_raw;
	LCP1_IO.VMB.VTB[m].DataNull							:= VMB1[m].DataNull; 
	LCP1_IO.VMB.VTB[m].LossVoltTransBoard				:= VMB1[m].LossVoltMonitorBoard;			
	
	VMB2[m] ( CapRaw := LCP2_IO.VMB.VTB[m].CapRaw );		
	LCP2_IO.VMB.VTB[m].BateryLow 						:= VMB2[m].BatteryLow;
	LCP2_IO.VMB.VTB[m].VoltageReading_raw				:= VMB2[m].VoltageReading_raw;
	LCP2_IO.VMB.VTB[m].DataNull							:= VMB2[m].DataNull; 
	LCP2_IO.VMB.VTB[m].LossVoltTransBoard				:= VMB2[m].LossVoltMonitorBoard;
END_FOR

//status - add VM.VTB to alarms.
(*
LCP1_IO.Segment[1].Module[1].VTB[1].BateryLow			:= LCP1_IO.VMB.VTB[0].BateryLow;
LCP1_IO.Segment[1].Module[1].VTB[1].DataNull 			:= LCP1_IO.VMB.VTB[0].DataNull;
LCP1_IO.Segment[1].Module[1].VTB[1].LossVoltTransBoard 	:= LCP1_IO.VMB.VTB[0].LossVoltTransBoard;
LCP1_IO.Segment[1].Module[1].VTB[2].BateryLow			:= LCP1_IO.VMB.VTB[1].BateryLow;
LCP1_IO.Segment[1].Module[1].VTB[2].DataNull			:= LCP1_IO.VMB.VTB[1].DataNull;
LCP1_IO.Segment[1].Module[1].VTB[2].LossVoltTransBoard	:= LCP1_IO.VMB.VTB[1].LossVoltTransBoard;

LCP1_IO.Segment[1].Module[2].VTB[1].BateryLow			:= LCP1_IO.VMB.VTB[2].BateryLow;
LCP1_IO.Segment[1].Module[2].VTB[1].DataNull			:= LCP1_IO.VMB.VTB[2].DataNull;
LCP1_IO.Segment[1].Module[2].VTB[1].LossVoltTransBoard	:= LCP1_IO.VMB.VTB[2].LossVoltTransBoard;
LCP1_IO.Segment[1].Module[2].VTB[2].BateryLow			:= LCP1_IO.VMB.VTB[3].BateryLow;
LCP1_IO.Segment[1].Module[2].VTB[2].DataNull			:= LCP1_IO.VMB.VTB[3].DataNull;
LCP1_IO.Segment[1].Module[2].VTB[2].LossVoltTransBoard	:= LCP1_IO.VMB.VTB[3].LossVoltTransBoard;

LCP1_IO.Segment[1].Module[3].VTB[1].BateryLow			:= LCP1_IO.VMB.VTB[4].BateryLow;
LCP1_IO.Segment[1].Module[3].VTB[1].DataNull			:= LCP1_IO.VMB.VTB[4].DataNull;
LCP1_IO.Segment[1].Module[3].VTB[1].LossVoltTransBoard	:= LCP1_IO.VMB.VTB[4].LossVoltTransBoard;
LCP1_IO.Segment[1].Module[3].VTB[2].BateryLow			:= LCP1_IO.VMB.VTB[5].BateryLow;
LCP1_IO.Segment[1].Module[3].VTB[2].DataNull			:= LCP1_IO.VMB.VTB[5].DataNull;
LCP1_IO.Segment[1].Module[3].VTB[2].LossVoltTransBoard	:= LCP1_IO.VMB.VTB[5].LossVoltTransBoard;

LCP1_IO.Segment[2].Module[4].VTB[1].BateryLow			:= LCP1_IO.VMB.VTB[6].BateryLow;
LCP1_IO.Segment[2].Module[4].VTB[1].DataNull			:= LCP1_IO.VMB.VTB[6].DataNull;
LCP1_IO.Segment[2].Module[4].VTB[1].LossVoltTransBoard	:= LCP1_IO.VMB.VTB[6].LossVoltTransBoard;
LCP1_IO.Segment[2].Module[4].VTB[2].BateryLow			:= LCP1_IO.VMB.VTB[7].BateryLow;
LCP1_IO.Segment[2].Module[4].VTB[2].DataNull			:= LCP1_IO.VMB.VTB[7].DataNull;
LCP1_IO.Segment[2].Module[4].VTB[2].LossVoltTransBoard	:= LCP1_IO.VMB.VTB[7].LossVoltTransBoard;

LCP1_IO.Segment[2].Module[5].VTB[1].BateryLow			:= LCP1_IO.VMB.VTB[8].BateryLow;
LCP1_IO.Segment[2].Module[5].VTB[1].DataNull			:= LCP1_IO.VMB.VTB[8].DataNull;
LCP1_IO.Segment[2].Module[5].VTB[1].LossVoltTransBoard	:= LCP1_IO.VMB.VTB[8].LossVoltTransBoard;
LCP1_IO.Segment[2].Module[5].VTB[2].BateryLow			:= LCP1_IO.VMB.VTB[9].BateryLow;
LCP1_IO.Segment[2].Module[5].VTB[2].DataNull			:= LCP1_IO.VMB.VTB[9].DataNull;
LCP1_IO.Segment[2].Module[5].VTB[2].LossVoltTransBoard	:= LCP1_IO.VMB.VTB[9].LossVoltTransBoard;
*)
//FOR i := 1 TO 3 BY 1 DO //segment 1 - 3
(*	IF i = 1 THEN 
		IF p > 0 THEN
			p := -3;
		END_IF 
		p := p + 1;
		j := p + q;	
		FOR k := 1 TO 2 BY 1 DO 		 
			//n vtb 0-17
			n := k + j + p; //
			LCP1_IO.Segment[i].Module[j].VoltageFeedback_raw[k] := LCP1_IO.VMB.VTB[n].VoltageReading_raw;
		END_FOR
	END_IF;
	*)
//END_FOR
(*
CASE eVoltFB OF
	E_VoltFB.seg1:
		i := 1;
		FOR j := 1 TO	3 BY 1 DO //module 1 -9			
			IF p > 0 THEN
				p := -3;
			END_IF 
			p := p + 1;
			j := p + q;	

			FOR k := 1 TO 2 BY 1 DO 		 
				//n vtb 0-17
				n := k + j + p; //
				LCP1_IO.Segment[i].Module[j].VoltageFeedback_raw[k] := LCP1_IO.VMB.VTB[n].VoltageReading_raw;
			END_FOR
			i := i +1;
			eVoltFB := E_VoltFB.seg2;
		END_FOR	
	E_VoltFB.seg2:
		IF p > 3 THEN
			p := 0;
		END_IF 
		p := p + 1;
		j := p + q;	

		FOR k := 1 TO 2 BY 1 DO 		 
				//n vtb 0-17
				n := k + j + p; //
				LCP1_IO.Segment[i].Module[j].VoltageFeedback_raw[k] := LCP1_IO.VMB.VTB[n].VoltageReading_raw;
		END_FOR
		i := i + 1;
		eVoltFB := E_VoltFB.seg3;
	E_VoltFB.seg3:
			IF p > 6 THEN
				p := 3;
			END_IF 
			p := p + 1;
			j := p + q;	

			FOR k := 1 TO 2 BY 1 DO 		 
				//n vtb 0-17
				n := k + j + p; //
				LCP1_IO.Segment[i].Module[j].VoltageFeedback_raw[k] := LCP1_IO.VMB.VTB[n].VoltageReading_raw;
			END_FOR
			i := i + 1;
			eVoltFB := E_VoltFB.seg3;
END_CASE
*)

LCP1_IO.Segment[1].Module[1].VoltageFeedback_raw[1] := LCP1_IO.VMB.VTB[0].VoltageReading_raw;
LCP1_IO.Segment[1].Module[1].VoltageFeedback_raw[2] := LCP1_IO.VMB.VTB[1].VoltageReading_raw;
LCP1_IO.Segment[1].Module[2].VoltageFeedback_raw[1] := LCP1_IO.VMB.VTB[2].VoltageReading_raw;
LCP1_IO.Segment[1].Module[2].VoltageFeedback_raw[2] := LCP1_IO.VMB.VTB[3].VoltageReading_raw;
LCP1_IO.Segment[1].Module[3].VoltageFeedback_raw[1] := LCP1_IO.VMB.VTB[4].VoltageReading_raw;
LCP1_IO.Segment[1].Module[3].VoltageFeedback_raw[2] := LCP1_IO.VMB.VTB[5].VoltageReading_raw;
LCP1_IO.Segment[2].Module[4].VoltageFeedback_raw[1] := LCP1_IO.VMB.VTB[6].VoltageReading_raw;
LCP1_IO.Segment[2].Module[4].VoltageFeedback_raw[2] := LCP1_IO.VMB.VTB[7].VoltageReading_raw;
LCP1_IO.Segment[2].Module[5].VoltageFeedback_raw[1] := LCP1_IO.VMB.VTB[8].VoltageReading_raw;
LCP1_IO.Segment[2].Module[5].VoltageFeedback_raw[2] := LCP1_IO.VMB.VTB[9].VoltageReading_raw;
LCP1_IO.Segment[2].Module[6].VoltageFeedback_raw[1] := LCP1_IO.VMB.VTB[10].VoltageReading_raw;
LCP1_IO.Segment[2].Module[6].VoltageFeedback_raw[2] := LCP1_IO.VMB.VTB[11].VoltageReading_raw;
LCP1_IO.Segment[3].Module[7].VoltageFeedback_raw[1] := LCP1_IO.VMB.VTB[12].VoltageReading_raw;
LCP1_IO.Segment[3].Module[7].VoltageFeedback_raw[2] := LCP1_IO.VMB.VTB[13].VoltageReading_raw;
LCP1_IO.Segment[3].Module[8].VoltageFeedback_raw[1] := LCP1_IO.VMB.VTB[14].VoltageReading_raw;
LCP1_IO.Segment[3].Module[8].VoltageFeedback_raw[2] := LCP1_IO.VMB.VTB[15].VoltageReading_raw;
LCP1_IO.Segment[3].Module[9].VoltageFeedback_raw[1] := LCP1_IO.VMB.VTB[16].VoltageReading_raw;
LCP1_IO.Segment[3].Module[9].VoltageFeedback_raw[2] := LCP1_IO.VMB.VTB[17].VoltageReading_raw;

LCP2_IO.Segment[4].Module[1].VoltageFeedback_raw[1] := LCP2_IO.VMB.VTB[0].VoltageReading_raw;
LCP2_IO.Segment[4].Module[1].VoltageFeedback_raw[2] := LCP2_IO.VMB.VTB[1].VoltageReading_raw;
LCP2_IO.Segment[4].Module[2].VoltageFeedback_raw[1] := LCP2_IO.VMB.VTB[2].VoltageReading_raw;
LCP2_IO.Segment[4].Module[2].VoltageFeedback_raw[2] := LCP2_IO.VMB.VTB[3].VoltageReading_raw;
LCP2_IO.Segment[4].Module[3].VoltageFeedback_raw[1] := LCP2_IO.VMB.VTB[4].VoltageReading_raw;
LCP2_IO.Segment[4].Module[3].VoltageFeedback_raw[2] := LCP2_IO.VMB.VTB[5].VoltageReading_raw;
LCP2_IO.Segment[5].Module[4].VoltageFeedback_raw[1] := LCP2_IO.VMB.VTB[6].VoltageReading_raw;
LCP2_IO.Segment[5].Module[4].VoltageFeedback_raw[2] := LCP2_IO.VMB.VTB[7].VoltageReading_raw;
LCP2_IO.Segment[5].Module[5].VoltageFeedback_raw[1] := LCP2_IO.VMB.VTB[8].VoltageReading_raw;
LCP2_IO.Segment[5].Module[5].VoltageFeedback_raw[2] := LCP2_IO.VMB.VTB[9].VoltageReading_raw;
LCP2_IO.Segment[5].Module[6].VoltageFeedback_raw[1] := LCP2_IO.VMB.VTB[10].VoltageReading_raw;
LCP2_IO.Segment[5].Module[6].VoltageFeedback_raw[2] := LCP2_IO.VMB.VTB[11].VoltageReading_raw;
LCP2_IO.Segment[6].Module[7].VoltageFeedback_raw[1] := LCP2_IO.VMB.VTB[12].VoltageReading_raw;
LCP2_IO.Segment[6].Module[7].VoltageFeedback_raw[2] := LCP2_IO.VMB.VTB[13].VoltageReading_raw;
LCP2_IO.Segment[6].Module[8].VoltageFeedback_raw[1] := LCP2_IO.VMB.VTB[14].VoltageReading_raw;
LCP2_IO.Segment[6].Module[8].VoltageFeedback_raw[2] := LCP2_IO.VMB.VTB[15].VoltageReading_raw;
LCP2_IO.Segment[6].Module[9].VoltageFeedback_raw[1] := LCP2_IO.VMB.VTB[16].VoltageReading_raw;
LCP2_IO.Segment[6].Module[9].VoltageFeedback_raw[2] := LCP2_IO.VMB.VTB[17].VoltageReading_raw;



IF i > 3 THEN 
	i := 1;
END_IF

IF j > 9 THEN 
	j := 1;
END_IF

IF k > 2 THEN 
	k := 1;
END_IF

IF m > 17 THEN
	m := 0;
END_IF


IF p >= 7 THEN
	p := -3;
END_IF

END_PROGRAM

// ---- POUs/Sequence.TcPOU
PROGRAM Sequence
VAR
	eState : E_State;
	
	ChargeRlyDelayON_Timer  : TON;
	ChargeRlyDelayDONE		: BOOL;
	ChargeRlyDelayON_PT		: TIME := T#250MS; //used for delay close and delay open for safe mode
	AbortPSnRlyDelay_Timer	: TON;
	AbortPSnRlyDelay_PT		: TIME := T#5MS; //defualt is 5ms
	AbortPSnRlyDelayDONE	: BOOL;
	ChargeCompleted			: BOOL;
	ChargingRunOutTMR_TON	: TON;
	ChargingRunOutTMR_ET	: TIME;
	ChargedRunOutTMR_TON	: TON;
	ChargedRunOutTMR_ET		: TIME;
	FireToSafeDelayTMR_TON	: TON;
	FireToSafeDelayTMR_PT	: TIME := T#5S;
	FireToSafeDelayTMR_ET	: TIME;
	FirePBpressed			: BOOL := FALSE;
	ShotFired				: BOOL := FALSE;
	
	ShotTrigDelayTMR_TON	: LTON;
	ShotTrigDelayTMR_PT		: LTIME := LTIME#10US;
	ShotTrigDelayTMR_ET		: LTIME;
	
	ShotTrigPulseTMR_TON	: LTON;
	ShotTrigPulseTMR_PT		: LTIME := LTIME#1S + ShotTrigDelayTMR_PT;
	ShotTrigPulseTMR_ET		: LTIME;
		
	ScopeTrigPulseTMR_TON	: TON;
	ScopeTrigPulseTMR_PT	: TIME := T#10MS;
	ScopeTrigPulseTMR_ET	: TIME;
	
	DumpingRunOutTMR_TON 	: TON;
	DumpingRunOutTMR_PT		: TIME := T#10S;
	DumpingRunOutTMR_ET		: TIME;
	LocalDumpActive			: BOOL := FALSE;

	StartChargingBroadcast	: BOOL := FALSE;
	StartCharger			: ARRAY[1..7] OF BOOL;

	ChargeTimeFinished		: BOOL;
	StartCharWarningTMR_TON : TON;
	StartCharWarningTMR_PT	: TIME := T#5S;
	StartCharWarningTMR_ET	: TIME;
	ChargeDelayStart		: BOOL := FALSE;
	
	DumpRlyDelayTMR_TON		: TON;
	DumpRlyDelay_PT			: TIME := T#250MS;
	DumpRlyDelay_ET			: TIME;
	
	i						: INT := 1; //1-7 chargers
	j						: INT := 1; //1-8 Shaft ramp dump rly
	k						: INT := 1; //1-9
	m						: INT := 1; //4-6
	n 						: INT := 7;
	CompDumpStagger			: Stagger_FB;
	SRDumpStagger			: Stagger_FB;
END_VAR

//Critical Delay Time
HMI_DB.ChargerHVOFF_rlyDelayPT := INT_TO_TIME(HMI_DB.ChargerHVOFF_rlyDelayPT_INT);
AbortPSnRlyDelay_PT := HMI_DB.ChargerHVOFF_rlyDelayPT;

//hv output delay
HMI_DB.HVONdelayPT := INT_TO_TIME (HMI_DB.HVONdelayPT_INT);
ChargeRlyDelayON_PT := HMI_DB.HVONdelayPT;

//runout timer
HMI_DB.RunOutTMR_PT := DINT_TO_TIME (HMI_DB.RunOutTMR_PT_INT*1000);
HMI_DB.RunOutTMR_elapse := (TIME_TO_DINT (HMI_DB.RunOutTMR_PT - ChargedRunOutTMR_TON.ET))/1000;
HMI_DB.ChargingRunOutTMR_elapse := TIME_TO_INT(ChargingRunOutTMR_TON.PT/1000 - ChargingRunOutTMR_TON.ET/1000);

//charge realy timer 
ChargeRlyDelayON_Timer(PT := ChargeRlyDelayON_PT);

//reset timer
IF eState <> E_State.CHARGING THEN 
	ChargingRunOutTMR_TON (IN := FALSE);
	//LCP1_IO.Segment[1].Module[1].ModuleCharged := FALSE; //for status light only

	FOR i := 1 TO n BY 1 DO
		ChargeTime_DB.ChargerDelay_TON[i] (IN := FALSE, PT := ChargeTime_DB.ChargerDelay_PT[i], ET => ChargeTime_DB.ChargerDelay_ET[i]);
		ChargeTime_DB.ChargingTimeElapse_TON[i].IN := FALSE;
		ChargeRlyDelayON_Timer (IN := FALSE);
	END_FOR;
	ChargeTime_DB.PreFormChargeTime_TON (IN := FALSE, PT := ChargeTime_DB.PreFormChargeTime_PT, ET => ChargeTime_DB.PreFormChargeTime_ET);
	ChargeTime_DB.PreFormChargingTimeElapse_TON.IN := FALSE;
END_IF

IF eState <> E_State.CHARGECOMPLETE THEN 
	//LCP1_IO.Segment[1].Module[1].ModuleCharged := FALSE; //for status light only
	ChargedRunOutTMR_TON (IN := FALSE); // only needed in charge complete
END_IF

IF HMI_DB.HMI_ManualModeSelected = TRUE AND eState = E_State.SAFE (*AND ChargeDelayStart = FALSE *)THEN //added charge delay start
	eState := E_State.ManualMode;
END_IF

IF eState = E_State.CHARGING OR eState = E_State.CHARGECOMPLETE OR eState = E_State.ABORT (*OR ChargeDelayStart = TRUE*) THEN //added charge delay start
	HMI_DB.HMI_ManualModeSelected := FALSE;
END_IF

IF eState <> E_State.ManualMode THEN
	HMI_DB.CloseChargeRlySW := FALSE;
	HMI_DB.OpenDumpRlySW := FALSE;
	HMI_DB.TurnChrgHVonSW := FALSE;
	HMI_DB.TurnChrgInhibitOffSW := FALSE;
	HMI_DB.TurnOnShotTrigSW := FALSE;
	HMI_DB.TurnOnChargeAlarm := FALSE;
END_IF

IF HMI_DB.DumpPB = TRUE THEN  //although will bring the state out of abort, it will go back to abort if faults are not clear.
	eState := E_State.DUMPING;
	ELSIF HMI_DB.AbortPB = TRUE OR Trips_DB.TimerRunOutON = TRUE THEN 
		eState := E_State.ABORT;
	//	ELSE
	//		eState := E_State.SAFE;
		END_IF;
		


CASE eState OF 
	//Safe OR IDLE
	E_State.SAFE:
		ChargeCompleted := FALSE;
		FirePBpressed := FALSE;
		FireToSafeDelayTMR_TON (IN := FALSE);
		ChargeRlyDelayON_Timer(IN:= FALSE);
		ChargeTime_DB.LongestChargeTime_TON (IN := FALSE); //reset timer
		ChargeTimeFinished := FALSE; //reset chargetime done bit
		ShotTrigDelayTMR_TON (IN := FALSE, PT := ShotTrigDelayTMR_PT, ET => ShotTrigDelayTMR_ET);
		ScopeTrigPulseTMR_TON (IN := FALSE, PT := ScopeTrigPulseTMR_PT, ET => ScopeTrigPulseTMR_ET);
		ShotTrigPulseTMR_TON (IN := FALSE, PT := ShotTrigPulseTMR_PT, ET => ShotTrigPulseTMR_ET);
		
		LCP1_IO.Fire := FALSE; //turn off all firing triggers
		LCP2_IO.Fire := FALSE;
		
		
		(*	// might not have interlock	
		IF Permissives_DB.CageInterlockOK = TRUE AND HMI_DB.ArmTheCagePB = TRUE THEN 
			MCP_IO.EnergizeACKontactor := TRUE;
		END_IF;
		*)
		
		//TURN OFF ALL CHARGERS
		FOR i := 1 TO n BY 1 DO 
			MCP_IO.Charger[i].inhibit := TRUE; // inhibit = high, no output | inhibit = low, allows output
			MCP_IO.Charger[i].HV_ON := FALSE; 
			//MCP_IO.Charger[i].voltageSP := 0.001;
			StartCharger[i] := FALSE; // reset bit
			ChargeTimeFinished := FALSE;
			StartChargingBroadcast := FALSE;
			//reset charger delay timer
			ChargeTime_DB.ChargerDelay_TON[i] (IN := FALSE, PT := ChargeTime_DB.ChargerDelay_PT[i], ET => ChargeTime_DB.ChargerDelay_ET[i]);
			ChargeTime_DB.ChargingTimeElapse_TON[i] (IN := FALSE); 
		END_FOR;
		ChargingRunOutTMR_TON (IN := FALSE);
		ChargedRunOutTMR_TON (IN := FALSE);
		DumpingRunOutTMR_TON (IN := FALSE);
		
		ScopeTrigPulseTMR_TON (IN := FALSE);
		ShotTrigDelayTMR_TON (IN := FALSE);
		ShotTrigPulseTMR_TON (IN := FALSE);
		
	
		LCP1_IO.Segment[1].CloseChargeRly := FALSE;
		LCP1_IO.Segment[2].CloseChargeRly := FALSE;
		LCP1_IO.Segment[3].CloseChargeRly := FALSE;
		
		LCP2_IO.Segment[4].CloseChargeRly := FALSE;
		LCP2_IO.Segment[5].CloseChargeRly := FALSE;
		LCP2_IO.Segment[6].CloseChargeRly := FALSE;
 
		//reset stagger fg
		CompDumpStagger (start := FALSE, n := 6, reset := TRUE); 
		LCP1_IO.Segment[1].OpenModule1To3DumpRly := FALSE;
		LCP1_IO.Segment[2].OpenModule4To6DumpRly := FALSE;
		LCP1_IO.Segment[3].OpenModule7To9DumpRly := FALSE;
		
		LCP2_IO.Segment[4].OpenModule1To3DumpRly := FALSE;
		LCP2_IO.Segment[5].OpenModule4To6DumpRly := FALSE;
		LCP2_IO.Segment[6].OpenModule7To9DumpRly := FALSE;
		
		(*shaft ramp*)
		LCP3_IO.CloseSRChargeRly := FALSE;
		
		//reset shaft ramp stagger first
		SRDumpStagger (start := FALSE, n := 8, reset := TRUE);
		FOR j := 1 TO 8 BY 1 DO 
			LCP3_IO.OpenSRDumpRly[j] := FALSE;
		END_FOR;
		
		IF HMI_DB.ChargePB = TRUE (*AND MCP_IO.EnergizeACKontactor*) THEN //directly sent from LV 
			ChargeDelayStart := TRUE;
		ELSIF HMI_DB.DumpPB = TRUE THEN
				eState := E_State.DUMPING; 
		END_IF;
		
		IF ChargeDelayStart = TRUE THEN
			// turn on warning light  
			LCP1_IO.SegmentCharged := TRUE;
			LCP2_IO.SegmentCharged := TRUE;
			LCP3_IO.SegmentCharged := TRUE;
			StartCharWarningTMR_TON (IN := TRUE, PT := StartCharWarningTMR_PT, ET=> StartCharWarningTMR_ET);
		END_IF;
		
		IF StartCharWarningTMR_TON.Q = TRUE THEN 
			ChargeDelayStart := FALSE;
			StartCharWarningTMR_TON (IN := FALSE);
			eState := E_State.CHARGING;
		END_IF

	E_State.CHARGING:
		StartCharWarningTMR_TON (IN := FALSE, PT := StartCharWarningTMR_PT, ET=> StartCharWarningTMR_ET);
		ChargeDelayStart := FALSE;
		// turn on warning light  
		LCP1_IO.SegmentCharged := TRUE;
		LCP2_IO.SegmentCharged := TRUE;
		LCP3_IO.SegmentCharged := TRUE;
		
		FirePBpressed := FALSE;
		LCP1_IO.Fire := FALSE;
		LCP2_IO.Fire := FALSE;
		//start charging runout timer
		LCP1_IO.Segment[1].CloseChargeRly := TRUE;
		LCP1_IO.Segment[2].CloseChargeRly := TRUE;
		LCP1_IO.Segment[3].CloseChargeRly := TRUE;
		
		LCP2_IO.Segment[4].CloseChargeRly := TRUE;
		LCP2_IO.Segment[5].CloseChargeRly := TRUE;
		LCP2_IO.Segment[6].CloseChargeRly := TRUE;
		
		LCP3_IO.CloseSRChargeRly := TRUE;
		
		//stagger the relays - change the name later
		CompDumpStagger (start := TRUE, n := 6, reset := FALSE);
		//or make sure the turn reset on when turning off the dump relay outputs
		LCP1_IO.Segment[1].OpenModule1To3DumpRly := CompDumpStagger.OutputHi[1]; //turn output ON
		LCP1_IO.Segment[2].OpenModule4To6DumpRly := CompDumpStagger.OutputHi[2];
		LCP1_IO.Segment[3].OpenModule7To9DumpRly := CompDumpStagger.OutputHi[3];
		LCP2_IO.Segment[4].OpenModule1To3DumpRly := CompDumpStagger.OutputHi[4];
		LCP2_IO.Segment[5].OpenModule4To6DumpRly := CompDumpStagger.OutputHi[5];
		LCP2_IO.Segment[6].OpenModule7To9DumpRly := CompDumpStagger.OutputHi[6];
		
		IF CompDumpStagger.OutputHi[6] = TRUE THEN 
			CompDumpStagger.start := FALSE;
		END_IF
		
		//stagger the dump relay for shaft ramp - total 8 dump rly
		SRDumpStagger (start := TRUE, n := 8, reset := FALSE);
		//open shaft ramp dump relays
		FOR j := 1 TO 8 BY 1 DO 
			LCP3_IO.OpenSRDumpRly[j] := SRDumpStagger.OutputHi[j];
		END_FOR;
		
		IF SRDumpStagger.OutputHi[8] = TRUE THEN 
			SRDumpStagger.start := FALSE;
		END_IF
		
